# B&R Automation Studio project TD52 (part 20)

### rtmmacros.h
```c
/*
 * Copyright 1994-2005 The MathWorks, Inc.
 *
 * File: rtmmacros.h     $Revision: 1.6.4.9 $
 *
 * Abstract:
 * All our real-time simulation wrappers are setup to handle rtModel
 * objects. For targets that still use the SimStruct, this file
 * provides a mapping from the rtModel to the SimStruct. When all targets
 * use the rtModel, this file can be eliminated.
 */

#ifndef _RTW_HEADER_rtmmacros_h_
# define _RTW_HEADER_rtmmacros_h_

#define rtmGetBlkStateChange            ssGetBlkStateChange
#define rtmSetBlkStateChange            ssSetBlkStateChange
#define rtmGetChecksum0                 ssGetChecksum0
#define rtmSetChecksum0                 ssSetChecksum0
#define rtmGetChecksum1                 ssGetChecksum1
#define rtmSetChecksum1                 ssSetChecksum1
#define rtmGetChecksum2                 ssGetChecksum2
#define rtmSetChecksum2                 ssSetChecksum2
#define rtmGetChecksum3                 ssGetChecksum3
#define rtmSetChecksum3                 ssSetChecksum3
#define rtmGetNumSampleTimes            ssGetNumSampleTimes
#define rtmGetNumContStates             ssGetNumContStates
#define rtmGetContStates                ssGetContStates
#define rtmSetContStates                ssSetContStates
#define rtmIsContinuousTask             ssIsContinuousTask
#define rtmGetDerivCacheNeedsReset      ssGetDerivCacheNeedsReset
#define rtmSetDerivCacheNeedsReset      ssSetDerivCacheNeedsReset
#define rtmGetDiscStates                ssGetDiscStates
#define rtmSetDiscStates                ssSetDiscStates
#define rtmGetErrorStatus               ssGetErrorStatus
#define rtmSetErrorStatus               ssSetErrorStatus
#define rtmGetFixedStepSize             ssGetFixedStepSize
#define rtmSetFixedStepSize             ssSetFixedStepSize
#define rtmGetRTWLogInfo                ssGetRTWLogInfo
#define rtmSetRTWLogInfo                ssSetRTWLogInfo
#define rtmGetRTWExtModeInfo            ssGetRTWExtModeInfo
#define rtmSetRTWExtModeInfo            ssSetRTWExtModeInfo
#define rtmGetMaxNumMinSteps            ssGetMaxNumMinSteps
#define rtmSetMaxNumMinSteps            ssSetMaxNumMinSteps
#define rtmGetMaxStepSize               ssGetMaxStepSize
#define rtmSetMaxStepSize               ssSetMaxStepSize
#define rtmGetMinStepSize               ssGetMinStepSize
#define rtmSetMinStepSize               ssSetMinStepSize
#define rtmGetSolverMaxConsecutiveMinStep   ssGetSolverMaxConsecutiveMinStep
#define rtmSetSolverMaxConsecutiveMinStep   ssSetSolverMaxConsecutiveMinStep
#define rtmGetSolverZcThreshold         ssGetSolverZcThreshold
#define rtmSetSolverZcThreshold         ssSetSolverZcThreshold
#define rtmGetSolverConsecutiveZCsError     ssGetSolverConsecutiveZCsError
#define rtmSetSolverConsecutiveZCsError     ssSetSolverConsecutiveZCsError
#define rtmGetSolverZeroCrossAlgorithm  ssGetSolverZeroCrossAlgorithm
#define rtmSetSolverZeroCrossAlgorithm  ssSetSolverZeroCrossAlgorithm
#define rtmGetSolverShapePreserveControl   ssGetSolverShapePreserveControl
#define rtmSetSolverShapePreserveControl   ssSetSolverShapePreserveControl
#define rtmGetModelMappingInfo          ssGetModelMappingInfo
#define rtmSetModelMappingInfo          ssSetModelMappingInfo
#define rtmGetOffsetTimePtr             ssGetOffsetTimePtr
#define rtmSetOffsetTimePtr             ssSetOffsetTimePtr
#define rtmGetPerTaskSampleHitsPtr      ssGetPerTaskSampleHitsPtr
#define rtmSetPerTaskSampleHitsPtr      ssSetPerTaskSampleHitsPtr
#define rtmIsSampleHit                  ssIsSampleHit
#define rtmSetSampleHitInTask           ssSetSampleHitInTask
#define rtmGetSampleHitPtr              ssGetSampleHitPtr
#define rtmSetSampleHitPtr              ssSetSampleHitPtr
#define rtmGetSampleTime                ssGetSampleTime
#define rtmSetSampleTime                ssSetSampleTime
#define rtmGetSampleTimePtr             ssGetSampleTimePtr
#define rtmSetSampleTimePtr             ssSetSampleTimePtr
#define rtmGetSampleTimeTaskIDPtr       ssGetSampleTimeTaskIDPtr
#define rtmSetSampleTimeTaskIDPtr       ssSetSampleTimeTaskIDPtr
#define rtmGetSimMode                   ssGetSimMode
#define rtmSetSimMode                   ssSetSimMode
#define rtmGetSimTimeStep               ssGetSimTimeStep
#define rtmSetSimTimeStep               ssSetSimTimeStep
#define rtmGetSolverAbsTol              ssGetSolverAbsTol
#define rtmSetSolverAbsTol              ssSetSolverAbsTol
#define rtmGetSolverData                ssGetSolverData
#define rtmSetSolverData                ssSetSolverData
#define rtmGetSolverMaxOrder            ssGetSolverMaxOrder
#define rtmSetSolverMaxOrder            ssSetSolverMaxOrder
#define rtmGetSolverConsecutiveZCsStepRelTol   ssGetSolverConsecutiveZCsStepRelTol
#define rtmSetSolverConsecutiveZCsStepRelTol   ssSetSolverConsecutiveZCsStepRelTol
#define rtmGetSolverMaxConsecutiveZCs   ssGetSolverMaxConsecutiveZCs
#define rtmSetSolverMaxConsecutiveZCs   ssSetSolverMaxConsecutiveZCs
#define rtmGetSolverExtrapolationOrder  ssGetSolverExtrapolationOrder
#define rtmSetSolverExtrapolationOrder  ssSetSolverExtrapolationOrder
#define rtmGetSolverNumberNewtonIterations   ssGetSolverNumberNewtonIterations
#define rtmSetSolverNumberNewtonIterations   ssSetSolverNumberNewtonIterations
#define rtmGetSolverMode                ssGetSolverMode
#define rtmSetSolverMode                ssSetSolverMode
#define rtmGetSolverName                ssGetSolverName
#define rtmSetSolverName                ssSetSolverName
#define rtmGetSolverNeedsReset          ssGetSolverNeedsReset
#define rtmSetSolverNeedsReset          ssSetSolverNeedsReset
#define rtmGetSolverRefineFactor        ssGetSolverRefineFactor
#define rtmSetSolverRefineFactor        ssSetSolverRefineFactor
#define rtmGetSolverRelTol              ssGetSolverRelTol
#define rtmSetSolverRelTol              ssSetSolverRelTol
#define rtmGetSolverStopTime            ssGetSolverStopTime
#define rtmSetSolverStopTime            ssSetSolverStopTime
#define rtmGetSolverRobustResetMethod   ssGetSolverRobustResetMethod
#define rtmSetSolverRobustResetMethod   ssSetSolverRobustResetMethod
#define rtmIsSpecialSampleHit           ssIsSpecialSampleHit
#define rtmGetStepSize                  ssGetStepSize
#define rtmSetStepSize                  ssSetStepSize
#define rtmGetStopRequested             ssGetStopRequested
#define rtmSetStopRequested             ssSetStopRequested
#define rtmGetT                         ssGetT
#define rtmSetT                         ssSetT
#define rtmGetTFinal                    ssGetTFinal
#define rtmSetTFinal                    ssSetTFinal
#define rtmGetTPtr                      ssGetTPtr
#define rtmSetTPtr                      ssSetTPtr
#define rtmGetTStart                    ssGetTStart
#define rtmSetTStart                    ssSetTStart
#define rtmGetTaskTime                  ssGetTaskTime
#define rtmSetTaskTime                  ssSetTaskTime
#define rtmGetTimeOfLastOutput          ssGetTimeOfLastOutput
#define rtmSetTimeOfLastOutput          ssSetTimeOfLastOutput
#define rtmGetTimingData                ssGetTimingData
#define rtmSetTimingData                ssSetTimingData
#define rtmGetU                         ssGetU
#define rtmSetU                         ssSetU
#define rtmGetVariableStepSolver        ssGetVariableStepSolver
#define rtmSetVariableStepSolver        ssSetVariableStepSolver
#define rtmGetY                         ssGetY
#define rtmSetY                         ssSetY
#define rtmGetZCCacheNeedsReset         ssGetZCCacheNeedsReset
#define rtmSetZCCacheNeedsReset         ssSetZCCacheNeedsReset
#define rtmGetdX                        ssGetdX
#define rtmSetdX                        ssSetdX
#define rtmOutputs                      sfcnOutputs
#define rtmTerminate                    sfcnTerminate
#define rtmInitializeSampleTimes        sfcnInitializeSampleTimes
#define rtmInitializeSizes              sfcnInitializeSizes
#define rtmUpdate                       sfcnUpdate
#define rtmDerivatives                  sfcnDerivatives
#define rtmStart                        sfcnStart
#endif                                  /* _RTW_HEADER_rtmmacros_h_ */

/* [EOF] rtmmacros.h */
```

### rtsplntypes.h
```c
#ifndef RTSPLNTYPES_H
#define RTSPLNTYPES_H

/*
 * File: rtsplntypes.h
 *
 * Abstract:
 *
 *   Typedefs for spline lookup table algorithms.
 *
 *   Copyright 1994-2007 The MathWorks, Inc.
 *
 *   $Revision: 1.1.6.1 $
 *
 */

#include "rtwtypes.h"

/***************************************************************
 *                n-D Table Work Data Structures               *
 ***************************************************************/

typedef struct rt_LUTnWork_tag
{
    const uint32_T *m_dimSizes;
    void           *m_tableData;
    void           **m_bpDataSet;
    uint32_T       *m_bpIndex;
    void           *m_bpLambda;
    const uint32_T *m_maxIndex;
} rt_LUTnWork;

typedef struct rt_LUTSplineWork_tag
{
    rt_LUTnWork    *m_TWork;
    void           *m_yyA;
    void           *m_yyB;
    void           *m_yy2;
    void           *m_up;
    void           *m_y2;
    const uint32_T *m_numYWorkElts;
} rt_LUTSplineWork;

#endif  /* RTSPLNTYPES_H */
```

### rtw_capi.h
```c
/*
 * Copyright 1994-2008 The MathWorks, Inc.
 *
 * File: rtw_capi.h     $Revision $
 *
 * Abstract:
 *   Provides structure types and constants generated by CAPI.
 *   Macros for accessing the fields of the structures are also provided.
 *   This header file is included in MODEL_capi.c
 *
 */

#ifndef _RTW_CAPI_H_
# define _RTW_CAPI_H_

#include <rtwtypes.h>

#define SS_ENUM_TYPE (MAX_uint8_T-1)
#define SS_STRUCT    (MAX_uint8_T)
#define rt_offsetof(s,el) ((uint16_T)((char_T *)&((s *)0)->el - (char_T *)(s *)0))

/* Enumeration for fixed point scaling type*/
typedef enum {
  rtwCAPI_FIX_UNIFORM_SCALING,
  rtwCAPI_FIX_NONUNIFORM_SCALING,
  rtwCAPI_FIX_RESERVED
} rtwCAPI_FixPtScalingType;

/* Enumeration for data orientation */
typedef enum {
  rtwCAPI_SCALAR,
  rtwCAPI_VECTOR,
  rtwCAPI_MATRIX_ROW_MAJOR,
  rtwCAPI_MATRIX_COL_MAJOR,
  rtwCAPI_MATRIX_COL_MAJOR_ND
} rtwCAPI_Orientation;

/* Signals Structure */
/* Fields of this stucture can be used to monitor block output signals*/
typedef struct rtwCAPI_Signals_tag {
  uint_T    addrMapIndex;  /* index into the data address map                */
  uint_T    sysNum;        /* system identification number, where 0 = root   */
  const char_T *blockPath; /* block's full path name (RTW mangled version)   */
  const char_T *signalName;/* signal label (unmangled, NULL if not present)  */
  uint16_T  portNumber;    /* port number  (starts at 0)                     */
  uint16_T  dataTypeIndex; /* index into DataTypeMap, gives signal data type */
  uint16_T  dimIndex;      /* index into DimensionMap, gives signal dimension*/
  uint16_T  fxpIndex;      /* index into FixPtMap, gives Fixed point info    */
  uint8_T   sTimeIndex;    /* index into SampleTimeMap, gives Task info      */
} rtwCAPI_Signals;

/* Macros for accessing Signals structure fields */
/* bio is a pointer to array of Signals structures */
#define rtwCAPI_GetSignalAddrIdx(bio, i)       ((bio)[(i)].addrMapIndex)
#define rtwCAPI_GetSignalBlockPath(bio, i)     ((bio)[(i)].blockPath)
#define rtwCAPI_GetSignalName(bio, i)          ((bio)[(i)].signalName)
#define rtwCAPI_GetSignalPortNumber(bio, i)    ((bio)[(i)].portNumber)
#define rtwCAPI_GetSignalDataTypeIdx(bio, i)   ((bio)[(i)].dataTypeIndex)
#define rtwCAPI_GetSignalDimensionIdx(bio, i)  ((bio)[(i)].dimIndex)
#define rtwCAPI_GetSignalFixPtIdx(bio, i)      ((bio)[(i)].fxpIndex)
#define rtwCAPI_GetSignalSampleTimeIdx(bio, i) ((bio)[(i)].sTimeIndex)
#define rtwCAPI_GetSignalSysNum(bio, i)        ((bio)[(i)].sysNum)

/* BlockParameters Structure */
/* Fields of this structure can be used to monitor/modify block parameters */
typedef struct rtwCAPI_BlockParameters_tag {
  uint_T    addrMapIndex;  /* index into the data address map                */
  const char_T *blockPath; /* block's full path name (RTW mangled version)   */
  const char_T *paramName; /* parameter name                                 */
  uint16_T  dataTypeIndex; /* index into DataTypeMap, gives param data type  */
  uint16_T  dimIndex;      /* index into DimensionMap, gives param dimensions*/
  uint16_T  fxpIndex;      /* index into FixPtMap, gives Fixed point info    */
} rtwCAPI_BlockParameters;

/* Macros for accessing BlockParameter structure fields */
/* prm is a pointer to array of BlockParameter structures */
#define rtwCAPI_GetBlockParameterAddrIdx(prm, i)      ((prm)[(i)].addrMapIndex)
#define rtwCAPI_GetBlockParameterBlockPath(prm, i)    ((prm)[(i)].blockPath)
#define rtwCAPI_GetBlockParameterName(prm, i)         ((prm)[(i)].paramName)
#define rtwCAPI_GetBlockParameterDataTypeIdx(prm, i)  ((prm)[(i)].dataTypeIndex)
#define rtwCAPI_GetBlockParameterDimensionIdx(prm, i) ((prm)[(i)].dimIndex)
#define rtwCAPI_GetBlockParameterFixPtIdx(prm, i)     ((prm)[(i)].fxpIndex)

/* ModelParameter Structure */
/* Fields of this structure can be used to monitor/modify model parameters   *
 * When Inline Parameters is on, you can configure tunable block parameters  *
 * as model parameters.                                                      */
typedef struct rtwCAPI_ModelParameters_tag {
  uint_T    addrMapIndex;  /* index into the data address map                */
  const char_T   *varName; /* variable  name                                 */
  uint16_T  dataTypeIndex; /* index into DataTypeMap, gives param data type  */
  uint16_T  dimIndex;      /* index into DimensionMap, gives param dimensions*/
  uint16_T  fxpIndex;      /* index into FixPtMap, gives Fixed point info    */
} rtwCAPI_ModelParameters;

/* Macros for accessing ModelParameter structure fields */
/* prm is a pointer to array of ModelParameter structures */
#define rtwCAPI_GetModelParameterAddrIdx(prm, i)      ((prm)[(i)].addrMapIndex)
#define rtwCAPI_GetModelParameterName(prm, i)         ((prm)[(i)].varName)
#define rtwCAPI_GetModelParameterDataTypeIdx(prm, i)  ((prm)[(i)].dataTypeIndex)
#define rtwCAPI_GetModelParameterDimensionIdx(prm, i) ((prm)[(i)].dimIndex)
#define rtwCAPI_GetModelParameterFixPtIdx(prm, i)     ((prm)[(i)].fxpIndex)

/* rtwCAPI_States Structure */
/* Fields of this stucture can be used to monitor block States */
typedef struct rtwCAPI_States_tag {
  uint_T addrMapIndex;     /* index into the data address map                 */
  int_T  contStateStartIndex; /* starting index in the model's continuous     *
                               * state and state derivative vectors. This is  *
                               * set to -1 for discrete states                */
  const char_T *blockPath; /* block's full path name (RTW mangled version)    */
  const char_T *stateName; /* state name, Default:DWork/Cont State Identifier */
  const char_T *pathAlias; /* Alias block path */
  uint16_T  dWorkIndex;    /* Index into the Block DWork, 0 for cont. states  */
  uint16_T  dataTypeIndex; /* index into DataTypeMap, gives state data type   */
  uint16_T  dimIndex;      /* index into DimensionMap, gives state dimensions */
  uint16_T  fxpIndex;      /* index into FixPtMap, gives Fixed point info     */
  uint8_T   sTimeIndex;    /* index into SampleTimeMap, gives Task info       */
  uint8_T   isContinuous;  /* if the state is a Continuous state*/
} rtwCAPI_States;

/* Macros for accessing States structure fields */
/* bState is a pointer to array of States structures */
#define rtwCAPI_GetStateAddrIdx(bState, i)       ((bState)[(i)].addrMapIndex)
#define rtwCAPI_GetContStateStartIndex(bState, i) \
        ((bState)[(i)].contStateStartIndex)
#define rtwCAPI_GetStateBlockPath(bState, i)     ((bState)[(i)].blockPath)
#define rtwCAPI_GetStateName(bState, i)          ((bState)[(i)].stateName)
#define rtwCAPI_GetStatePathAlias(bState, i)     ((bState)[(i)].pathAlias)
#define rtwCAPI_GetStateDWorkIdx(bState, i)      ((bState)[(i)].dWorkIndex)
#define rtwCAPI_GetStateDataTypeIdx(bState, i)   ((bState)[(i)].dataTypeIndex)
#define rtwCAPI_GetStateDimensionIdx(bState, i)  ((bState)[(i)].dimIndex)
#define rtwCAPI_GetStateFixPtIndex(bState, i)    ((bState)[(i)].fxpIndex)
#define rtwCAPI_GetStateSampleTimeIdx(bState, i) ((bState)[(i)].sTimeIndex)
#define rtwCAPI_IsAContinuousState(bState, i)    ((bState)[(i)].isContinuous == 1)

/* DataTypeMap structure */
/* Members provide data type information of a signal or parameter */
typedef struct rtwCAPI_DataTypeMap_tag {
  const char_T *cDataName;   /* C language data type name                    */
  const char_T *mwDataName;  /* MathWorks data type, typedef in rtwtypes.h   */
  uint16_T      numElements; /* number of elements, 0 for non-structure data */
  uint16_T      elemMapIndex;/* index into the ElementMap, gives Bus Info    */
  uint16_T      dataSize;    /* data size in Bytes                           */
  uint8_T       slDataId;    /* enumerated data type from simstruc_types.h   */
  unsigned int  isComplex:1; /* is the data type complex (1=Complex, 0=Real) */
  unsigned int  isPointer:1; /* is data accessed Via Pointer (1=yes, 0= no)  */
} rtwCAPI_DataTypeMap;

/* Notes on rtwCAPI_DataTypeMap:
 * cDataName  - The ANSI C equivalent data type.
 *              For fixed point data
 *                  cDataName = the native integer equivalent
 *              For Complex data or non-virtual structures,
 *                  cDataName = "struct"
 * mwDataName - RTW defined data type. Typedef can be found in rtwtypes.h
 *              For fixed point data,
 *                  mwDataName = the integer type in which the data is stored.
 *                  Use rtwCAPI_FixPtMap to get slope & bias of the data.
 * numElements - Number of elements/members in the data type. If the data type
 *              represents a non-virtual structure (for e.g, bus structure),
 *              this field gives the number of elements in the structure.
 *              For non-structure data type, the default value is 0
 *              Complex data types are treated as non-structures
 * elemMapIndex - Index into the rtwCAPI_ElementMap which maps each of the
 *              element/member of a structure data type.
 * slDataId   - Enumerated Simulink Data type defined in simstruc_types.h.
 *              The enumerations are
 *                 o SS_DOUBLE
 *                 o SS_SINGLE
 *                 o SS_INT8
 *                 o SS_UINT8
 *                 o SS_INT16
 *                 o SS_UINT16
 *                 o SS_INT32
 *                 o SS_UINT32
 *                 o SS_BOOLEAN
 *                 o SS_ENUM_TYPE  (for enumerated data types)
 *                 o SS_STRUCT     (for non-virtual structures)
 *              For fixed point data:
 *                  slDataId = enumeration corresponding to the integer type
 *                             in which the data is stored
 *              For Complex data:
 *                  slDataId = enumeration corresponding to the data type of
 *                             the real part.
 * isComplex  - is the data type complex (1=Complex, 0=Real)
 * isPointer  - is data accessed Via Pointer (1=yes, 0= no)
 */

/* Macros for accessing DataTypeMap fields/members */
#define rtwCAPI_GetDataTypeCName(dTypeMap, i)       ((dTypeMap)[(i)].cDataName)
#define rtwCAPI_GetDataTypeMWName(dTypeMap, i)      ((dTypeMap)[(i)].mwDataName)
#define rtwCAPI_GetDataTypeNumElements(dTypeMap, i) ((dTypeMap)[(i)].numElements)
#define rtwCAPI_GetDataTypeElemMapIndex(dTypeMap,i) ((dTypeMap)[(i)].elemMapIndex)
#define rtwCAPI_GetDataTypeSLId(dTypeMap, i)        ((dTypeMap)[(i)].slDataId)
#define rtwCAPI_GetDataTypeSize(dTypeMap, i)        ((dTypeMap)[(i)].dataSize)
#define rtwCAPI_GetDataIsComplex(dTypeMap, i)       ((dTypeMap)[(i)].isComplex)
#define rtwCAPI_GetDataIsPointer(dTypeMap, i)       ((dTypeMap)[(i)].isPointer)

/* Macros for determining whether signals/states support MAT-File logging */
#define rtwCAPI_CanLogSignalToMATFile(dTypeMap, bio, i) \
    (rtwCAPI_GetDataTypeSLId(dTypeMap, rtwCAPI_GetSignalDataTypeIdx(bio, i))   < SS_NUM_BUILT_IN_DTYPE)
#define rtwCAPI_CanLogStateToMATFile(dTypeMap, bState, i) \
    (rtwCAPI_GetDataTypeSLId(dTypeMap, rtwCAPI_GetStateDataTypeIdx(bState, i)) < SS_NUM_BUILT_IN_DTYPE)

/* ElementMap structure */
/* Fields provide information on elements (fields) in Simulink Bus structure */
typedef struct rtwCAPI_ElementMap_tag {
  const char_T   *elementName;   /* name of the element                      */
  uint16_T  elementOffset; /* offset of the structure element in bytes       */
  uint16_T  dataTypeIndex; /* index into DataTypeMap, datatype of the element*/
  uint16_T  dimIndex;      /* index into DimensionMap, element's dimensions  */
  uint16_T  fxpIndex;      /* index into fixPtMap, fixed point information   */
} rtwCAPI_ElementMap;

/* Macros for accessing ElementMap fields */
#define rtwCAPI_GetElementName(elemMap, i)         ((elemMap)[(i)].elementName)
#define rtwCAPI_GetElementOffset(elemMap, i)       ((elemMap)[(i)].elementOffset)
#define rtwCAPI_GetElementDataTypeIdx(elemMap, i)  ((elemMap)[(i)].dataTypeIndex)
#define rtwCAPI_GetElementDimensionIdx(elemMap, i) ((elemMap)[(i)].dimIndex)
#define rtwCAPI_GetElementFixPtIdx(elemMap, i)     ((elemMap)[(i)].fxpIndex)

/* DimensionMap structure */
/* Fields provide dimensions of a signal or a parameter */
typedef struct rtwCAPI_DimensionMap_tag {
  rtwCAPI_Orientation orientation;
                                 /* orientation of data -scalar/vector/matrix/ND */
  uint_T    dimArrayIndex;       /* index into dimension array                   */
  uint8_T   numDims;             /* number of dimensions                         */
  uint_T    vardimsIndex;        /* index into vardims address array             */
} rtwCAPI_DimensionMap;

/* Macros for accessing DimensionMap fields */
#define rtwCAPI_GetOrientation(dimMap, i)    ((dimMap)[(i)].orientation)
#define rtwCAPI_GetDimArrayIndex(dimMap, i)  ((dimMap)[(i)].dimArrayIndex)
#define rtwCAPI_GetNumDims(dimMap, i)        ((dimMap)[(i)].numDims)
#define rtwCAPI_GetDimsIsVariable(vardimsAddrMap, dimMap, i) (vardimsAddrMap[(dimMap)[(i)].vardimsIndex] != NULL)

/* FixPtMap Structure */
/* Fields provide fixed point information of a signal or parameter */
typedef struct rtwCAPI_FixPtMap_tag {
  const void*       fracSlopePtr;   /* pointer to fractional slope value        */
  const void*       biasPtr;        /* pointer to bias value                    */
  rtwCAPI_FixPtScalingType scaleType;
                              /* scaling type - uniform/non-uniform       */
  uint8_T     wordLength;     /* number of bits required to store value   *
                               * In MATLAB, word length of the fi object  */
  int8_T      exponent;       /* exponent                                 */
  boolean_T   isSigned;       /* 1 = signed data, 0 = unsigned data       */
} rtwCAPI_FixPtMap;

/* Macros for accessing FixPtMap fields */
#define rtwCAPI_GetFxpFracSlopePtr(fxpMap, i) ((fxpMap)[(i)].fracSlopePtr)
#define rtwCAPI_GetFxpBiasPtr(fxpMap, i)      ((fxpMap)[(i)].biasPtr)
#define rtwCAPI_GetFxpScaling(fxpMap, i)      ((fxpMap)[(i)].scaleType)
#define rtwCAPI_GetFxpWordLength(fxpMap, i)   ((fxpMap)[(i)].wordLength)
#define rtwCAPI_GetFxpExponent(fxpMap, i)     ((fxpMap)[(i)].exponent)
#define rtwCAPI_GetFxpIsSigned(fxpMap, i)     ((fxpMap)[(i)].isSigned)

/* Macros to get the slope and bias values casted to DOUBLE */
#define rtwCAPI_GetFxpFracSlope(fxpMap, i) (*((real_T*) rtwCAPI_GetFxpFracSlopePtr(fxpMap,i)))
#define rtwCAPI_GetFxpBias(fxpMap, i)      (*((real_T*) rtwCAPI_GetFxpBiasPtr(fxpMap, i)))

/* SampleTimeMap Structure */
typedef struct rtwCAPI_SampleTimeMap_tag {
  const void*     samplePeriodPtr;  /* pointer to sample time period value       */
  const void*     sampleOffsetPtr;  /* pointer to sample time Offset value       */
  int8_T    tid;              /* task identifier                           */
  uint8_T   samplingMode;     /* 1 = FrameBased, 0 = SampleBased           */
} rtwCAPI_SampleTimeMap;

/* Macros for accessing SampleTimeMap fields */

#define rtwCAPI_GetSamplePeriodPtr(sampTimeMap, i) ((sampTimeMap)[(i)].samplePeriodPtr)
#define rtwCAPI_GetSampleOffsetPtr(sampTimeMap, i) ((sampTimeMap)[(i)].sampleOffsetPtr)
#define rtwCAPI_GetSampleTimeTID(sampTimeMap, i)   ((sampTimeMap)[(i)].tid)
#define rtwCAPI_GetSamplingMode(sampTimeMap, i)    ((sampTimeMap)[(i)].samplingMode)

/* Macros to get sample period and offset casted to DOUBLE */
#define rtwCAPI_GetSamplePeriod(sampTimeMap, i) (*((real_T *) rtwCAPI_GetSamplePeriodPtr(sampTimeMap, i)))
#define rtwCAPI_GetSampleOffset(sampTimeMap, i) (*((real_T *) rtwCAPI_GetSampleOffsetPtr(sampTimeMap, i)))

/* Macro to get the actual data address */
#define rtwCAPI_GetDataAddress(dataAddrMap,addrIdx) ((dataAddrMap)[(addrIdx)])

/* Macro to get the actual var dims address */
#define rtwCAPI_GetCurrentDimsAddr(vardimsAddrMap,dimMap,addrIdx) ((vardimsAddrMap)[(dimMap)[(addrIdx)].vardimsIndex])

#endif /* _RTW_CAPI_H_ */

/* EOF - rtw_capi.h */
```

### rtw_capi_examples.h
```c
/*
 * Copyright 2004 The MathWorks, Inc.
 *
 * File: rtw_capi_examples.h     $Revision: 1.1.4.2 $
 *
 * Abstract:
 *   Provides utility functions to traverse and access RTW generated C-API
 *   structures. The C-API structure types are provided in following 2 files.
 *
 *       matlabroot/rtw/c/src/rtw_capi.h & rtw_modelmap.h
 *
 *   The actual data structures are generated by code generator in
 *   <MODEL>_capi.c, where <MODEL> is the name of the model.
 *
 *   The functions provided in this file are
 *       capi_PrintModelParameter - Prints a model parameter value to STDOUT
 */

#ifndef __RTW_CAPI_EXAMPLES_H__
# define __RTW_CAPI_EXAMPLES_H__

#include <stdio.h>
#include <assert.h>
#include <math.h>
#include "rtwtypes.h"
#include "rtw_modelmap.h"

#ifdef __cplusplus
extern "C" {
#endif

extern void capi_PrintModelParameter(rtwCAPI_ModelMappingInfo* capiMap,
                                     uint_T                    paramIdx);

extern void capi_PrintParameter(const char_T*  paramName,
                                void*          paramAddress,
                                uint8_T        slDataId,
                                unsigned short isComplex,
                                uint_T*        actDims,
                                uint_T         numDims,
                                real_T         slope,
                                real_T         bias);

extern int_T capi_ModifyModelParameter(rtwCAPI_ModelMappingInfo* capiMap,
                                       uint_T                    paramIdx,
                                       void*                     newParam);

extern int_T capi_ModifyParameter(void                 *_param,
                                  void                 *_newParam,
                                  rtwCAPI_Orientation  orientation,
                                  uint_T               *dims,
                                  uint8_T              nDims,
                                  uint8_T              slDataType,
                                  unsigned short       isComplex);

#ifdef __cplusplus
}
#endif

#endif

/* EOF - rtw_capi_example.h */
```

### rtw_continuous.h
```c
/*
 * Copyright 1990-2009 The MathWorks, Inc.
 *
 * File: rtw_continuous.h     $Revision: 1.1.6.3 $
 *
 * Abstract:
 *   Type definitions for continuous-time support.
 *
 */

#ifndef __RTW_CONTINUOUS_H__
#define __RTW_CONTINUOUS_H__

/* For models registering MassMatrix */
typedef enum {
    SS_MATRIX_NONE,
    SS_MATRIX_CONSTANT,
    SS_MATRIX_TIMEDEP,
    SS_MATRIX_STATEDEP
} ssMatrixType;

typedef enum {
    SOLVER_MODE_AUTO,          /* only occurs in
                                  mdlInitializeSizes/mdlInitializeSampleTimes */
    SOLVER_MODE_SINGLETASKING,
    SOLVER_MODE_MULTITASKING
} SolverMode;

typedef enum {
    MINOR_TIME_STEP,
    MAJOR_TIME_STEP
} SimTimeStep;

/* =============================================================================
 * Model methods object
 * =============================================================================
 */
typedef void (*rtMdlInitializeSizesFcn)(void *rtModel);
typedef void (*rtMdlInitializeSampleTimesFcn)(void *rtModel);
typedef void (*rtMdlStartFcn)(void *rtModel);
typedef void (*rtMdlOutputsFcn)(void *rtModel, int_T tid);
typedef void (*rtMdlUpdateFcn)(void *rtModel, int_T tid);
typedef void (*rtMdlDerivativesFcn)(void *rtModel);
typedef void (*rtMdlProjectionFcn)(void *rtModel);
typedef void (*rtMdlMassMatrixFcn)(void *rtModel);
typedef void (*rtMdlForcingFunctionFcn)(void *rtModel);
typedef void (*rtMdlTerminateFcn)(void *rtModel);
#ifdef RT_MALLOC
typedef real_T (*rtMdlDiscreteEventsFcn)(void  *pModel,
                                         int_T  rtmNumSampTimes,
                                         void  *rtmTimingData,
                                         int_T  *rtmSampleHitPtr,
                                         int_T  *rtmPerTaskSampleHits);
#endif

typedef struct _RTWRTModelMethodsInfo_tag {
    void                          *rtModelPtr;
    rtMdlInitializeSizesFcn       rtmInitSizesFcn;
    rtMdlInitializeSampleTimesFcn rtmInitSampTimesFcn;
    rtMdlStartFcn                 rtmStartFcn;
    rtMdlOutputsFcn               rtmOutputsFcn;
    rtMdlUpdateFcn                rtmUpdateFcn;
    rtMdlDerivativesFcn           rtmDervisFcn;
    rtMdlProjectionFcn            rtmProjectionFcn;
    rtMdlMassMatrixFcn            rtmMassMatrixFcn;
    rtMdlForcingFunctionFcn       rtmForcingFunctionFcn;
    rtMdlTerminateFcn             rtmTerminateFcn;
#ifdef  RT_MALLOC
    rtMdlDiscreteEventsFcn        rtmDiscreteEventsFcn;
#endif
} RTWRTModelMethodsInfo;

#define rtmiSetRTModelPtr(M,rtmp) ((M).rtModelPtr = (rtmp))
#define rtmiGetRTModelPtr(M)      (M).rtModelPtr

#define rtmiSetInitSizesFcn(M,fp) \
  ((M).rtmInitSizesFcn = ((rtMdlInitializeSizesFcn)(fp)))
#define rtmiSetInitSampTimesFcn(M,fp) \
  ((M).rtmInitSampTimesFcn = ((rtMdlInitializeSampleTimesFcn)(fp)))
#define rtmiSetStartFcn(M,fp) \
  ((M).rtmStartFcn = ((rtMdlStartFcn)(fp)))
#define rtmiSetOutputsFcn(M,fp) \
  ((M).rtmOutputsFcn = ((rtMdlOutputsFcn)(fp)))
#define rtmiSetUpdateFcn(M,fp) \
  ((M).rtmUpdateFcn = ((rtMdlUpdateFcn)(fp)))
#define rtmiSetDervisFcn(M,fp) \
  ((M).rtmDervisFcn = ((rtMdlDerivativesFcn)(fp)))
#define rtmiSetProjectionFcn(M,fp) \
  ((M).rtmProjectionFcn = ((rtMdlProjectionFcn)(fp)))
#define rtmiSetMassMatrixFcn(M,fp) \
  ((M).rtmMassMatrixFcn = ((rtMdlMassMatrixFcn)(fp)))
#define rtmiSetForcingFunctionFcn(M,fp) \
  ((M).rtmForcingFunctionFcn = ((rtMdlForcingFunctionFcn)(fp)))
#define rtmiSetTerminateFcn(M,fp) \
  ((M).rtmTerminateFcn = ((rtMdlTerminateFcn)(fp)))
#ifdef  RT_MALLOC
#define rtmiSetDiscreteEventsFcn(M,fp) \
  ((M).rtmDiscreteEventsFcn = ((rtMdlDiscreteEventsFcn)(fp)))
#endif

#define rtmiInitializeSizes(M)                  \
    ((*(M).rtmInitSizesFcn)((M).rtModelPtr))
#define rtmiInitializeSampleTimes(M)                    \
    ((*(M).rtmInitSampTimesFcn)((M).rtModelPtr))
#define rtmiStart(M) \
    ((*(M).rtmStartFcn)((M).rtModelPtr))
#define rtmiOutputs(M, tid) \
    ((*(M).rtmOutputsFcn)((M).rtModelPtr,tid))
#define rtmiUpdate(M, tid) \
    ((*(M).rtmUpdateFcn)((M).rtModelPtr,tid))
#define rtmiDerivatives(M) \
    ((*(M).rtmDervisFcn)((M).rtModelPtr))
#define rtmiProjection(M) \
    ((*(M).rtmProjectionFcn)((M).rtModelPtr))
#define rtmiMassMatrix(M) \
    ((*(M).rtmMassMatrixFcn)((M).rtModelPtr))
#define rtmiForcingFunction(M) \
    ((*(M).rtmForcingFunctionFcn)((M).rtModelPtr))
#define rtmiTerminate(M) \
    ((*(M).rtmTerminateFcn)((M).rtModelPtr))
#ifdef  RT_MALLOC
#define rtmiDiscreteEvents(M,x1,x2,x3,x4)                               \
    ((*(M).rtmDiscreteEventsFcn)((M).rtModelPtr,(x1),(x2),(x3),(x4)))
#endif
#endif /* __RTW_CONTINUOUS_H__ */
```

### rtw_extmode.h
```c
/*
 * Copyright 1990-2008 The MathWorks, Inc.
 *
 * File: rtw_extmode.h     $Revision: 1.1.6.3 $
 *
 * Abstract:
 *   Type definitions for Simulink External Mode support.
 */

#ifndef __RTW_EXTMODE_H__
#define __RTW_EXTMODE_H__

/* =============================================================================
 * External mode object
 * =============================================================================
 */
typedef struct _RTWExtModeInfo_tag {

    void *subSysActiveVectorAddr;  /* Array of addresses pointing to
                                    * the active vector slots for sub-systems.
                                    * Sub-systems store information about their
                                    * state in their extmode active vector.
                                    */
    uint32_T *checksumsPtr;        /* Pointer to the model's checksums array
                                    */
    const void **mdlMappingInfoPtr;/* Pointer to the model's mapping info
                                    * pointer
                                    */

#if !defined(ENABLE_SLEXEC_SSBRIDGE)
    void       *tPtr;              /* Copy of model's time pointer */
#else
    void* simStruct;
#endif

    int32_T tFinalTicks;           /* Used with integer only code, holds the
                                    * number of base rate ticks representing
                                    * the final time (final time in seconds
                                    * divided by base rate step size).
                                    */

} RTWExtModeInfo;

/* gnat 3.12a2 doesn't like use "/" as line continuation here */
#define rteiSetSubSystemActiveVectorAddresses(E,addr) ((E)->subSysActiveVectorAddr = ((void *)addr))
#define rteiGetSubSystemActiveVectorAddresses(E)    ((E)->subSysActiveVectorAddr)
#define rteiGetAddrOfSubSystemActiveVector(E,idx)   ((int8_T*)((int8_T**)((E)->subSysActiveVectorAddr))[idx])

#define rteiSetModelMappingInfoPtr(E,mip) ((E)->mdlMappingInfoPtr = (mip))
#define rteiGetModelMappingInfo(E) (*((E)->mdlMappingInfoPtr))

#define rteiSetChecksumsPtr(E,cp) ((E)->checksumsPtr = (cp))
#define rteiGetChecksum0(E) (E)->checksumsPtr[0]
#define rteiGetChecksum1(E) (E)->checksumsPtr[1]
#define rteiGetChecksum2(E) (E)->checksumsPtr[2]
#define rteiGetChecksum3(E) (E)->checksumsPtr[3]

#if !defined(ENABLE_SLEXEC_SSBRIDGE)
# define rteiSetTPtr(E,p) ((E)->tPtr = (p))
# define rteiGetT(E)      ((time_T *)(E)->tPtr)[0]
#endif

#define rteiGetTFinalTicks(E) ((int32_T)((E)->tFinalTicks))
#define rteiGetPtrTFinalTicks(E) ((int32_T *)(&((E)->tFinalTicks)))

/*
 * UNUSED_PARAMETER(x)
 *   Used to specify that a function parameter (argument) is required but not
 *   accessed by the function body.
 */
#ifndef UNUSED_PARAMETER
# if defined(__LCC__)
#   define UNUSED_PARAMETER(x)  /* do nothing */
# else
/*
 * This is the semi-ANSI standard way of indicating that a
 * unused function parameter is required.
 */
#   define UNUSED_PARAMETER(x) (void) (x)
# endif
#endif

#endif /* __RTW_EXTMODE_H__ */
```

### rtw_linux.h
```c
#ifndef RTW_LINUX_H
#define RTW_LINUX_H

/*
 * Copyright 2011 The MathWorks, Inc.
 *
 * File: rtw_linux.h
 *
 * Abstract:
 *  Function prototypes and defines pthread mutex/semaphores
 */
#include <pthread.h>
#include <stdlib.h>
#include <semaphore.h>

#ifndef __USE_UNIX98
#define __USE_UNIX98
#endif

#ifdef __cplusplus
extern "C" {
#endif

extern void rtw_pthread_mutex_init( void** mutexDW );

#ifdef __cplusplus
}
#endif

#define rtw_pthread_mutex_lock( mutexDW ) \
    pthread_mutex_lock((pthread_mutex_t *)(mutexDW));

#define rtw_pthread_mutex_unlock( mutexDW ) \
    pthread_mutex_unlock((pthread_mutex_t *)(mutexDW));

#define rtw_pthread_mutex_destroy( mutexDW )      \
    pthread_mutex_destroy((pthread_mutex_t *)(mutexDW)); \
    free(mutexDW);

#define rtw_pthread_sem_create( semaphoreDW, initVal ) \
    *semaphoreDW = malloc(sizeof(sem_t));               \
    sem_init(*(semaphoreDW), 0, (initVal));

#define rtw_pthread_sem_wait( semaphoreDW ) \
    sem_wait(semaphoreDW);

#define rtw_pthread_sem_post( semaphoreDW ) \
    sem_post(semaphoreDW);

#define rtw_pthread_sem_destroy( semaphoreDW ) \
    sem_destroy(semaphoreDW);                   \
    free(semaphoreDW);

#endif /* RTW_LINUX_H */

/* LocalWords:  pthread
 */
```

### rtw_linux_mac.h
```c
#ifndef RTW_LINUX_MAC_H
#define RTW_LINUX_MAC_H

/*
 * Copyright 2011 The MathWorks, Inc.
 *
 * File: rtw_linux_mac.h
 *
 * Abstract:
 *  Function prototypes and defines pthread mutex/semaphores
 */
#ifdef __cplusplus
extern "C" {
#endif

#include <pthread.h>
#include <stdlib.h>
#include <semaphore.h>

#ifndef __USE_UNIX98
#define __USE_UNIX98
#endif

extern void rtw_pthread_mutex_init_mac( void** mutexDW );

#define rtw_pthread_mutex_lock_mac( mutexDW )                   \
    pthread_mutex_lock((pthread_mutex_t *)(mutexDW));

#define rtw_pthread_mutex_unlock_mac( mutexDW )                 \
    pthread_mutex_unlock((pthread_mutex_t *)(mutexDW));

#define rtw_pthread_mutex_destroy_mac( mutexDW )                \
    pthread_mutex_destroy((pthread_mutex_t *)(mutexDW));        \
    free(mutexDW);

extern void rtw_pthread_sem_create_mac( void** semaphoreDW1,
                                 void** semaphoreDW2,
                                 long initVal );

#define rtw_pthread_sem_wait_mac( semaphoreDW ) \
    sem_wait(semaphoreDW);

#define rtw_pthread_sem_post_mac( semaphoreDW ) \
    sem_post(semaphoreDW);

#define rtw_pthread_sem_destroy_mac( semaphoreDW ) \
    sem_unlink((char*)(semaphoreDW));              \
    free(semaphoreDW);

#ifdef __cplusplus
}
#endif

#endif /* RTW_LINUX_MAC_H */

/* LocalWords:  pthread
 */
```

### rtw_matlogging.h
```c
/*
 * Copyright 1990-2007 The MathWorks, Inc.
 *
 * File: rtw_matlogging.h     $Revision: 1.1.6.3 $
 *
 * Abstract:
 *   Type definitions for MAT-file logging support.
 */

#ifndef __RTW_MATLOGGING_H__
#define __RTW_MATLOGGING_H__

/*
 * The RTWLogSignalInfo and RTWLogInfo structures are for use by
 * the Real-Time Workshop and should not be used by S-functions.
 */
typedef const int8_T * const * LogSignalPtrsType;

#ifndef NO_FLOATS /* ERT integer-only */

typedef struct RTWLogDataTypeConvert_tag {

    int conversionNeeded;
    BuiltInDTypeId dataTypeIdLoggingTo;
    DTypeId        dataTypeIdOriginal;
    int            bitsPerChunk;
    int            numOfChunk;
    unsigned int   isSigned;
    real_T         fracSlope;
    int            fixedExp;
    real_T         bias;

} RTWLogDataTypeConvert;

typedef struct RTWLogSignalInfo_tag {
    int_T           numSignals;
    int_T          *numCols;
    int_T          *numDims;
    int_T          *dims;
    boolean_T      *isVarDims;       /* Dimension Mode: true -- VarDims / false -- fixed dims */
    void           **currSigDims;    /* current signal dimensions */
    int_T          *currSigDimsSize; /* Size of currSigDims in bytes */
    BuiltInDTypeId *dataTypes;
    int_T          *complexSignals;
    int_T          *frameData;

    union {
        const char_T** cptr;
        char_T**       ptr;
    } labels;

    char_T         *titles;
    int_T          *titleLengths;
    int_T          *plotStyles;

    union {
        const char_T** cptr;
        char_T**       ptr;
    } blockNames;

    union {
        const char_T** cptr;
        char_T**       ptr;
    } stateNames;

    boolean_T      *crossMdlRef;

    RTWLogDataTypeConvert *dataTypeConvert;

} RTWLogSignalInfo;

/* =============================================================================
 * Logging object
 * =============================================================================
 */
typedef struct _RTWLogInfo_tag {
  void              *logInfo;      /* Pointer to a book keeping structure    *
                                    * used in rtwlog.c                       */

  union {
      LogSignalPtrsType cptr; /* Pointers to the memory location    */
      int8_T**    ptr;        /* of the data to be logged into the  *
                               * states structure. Not used if      *
                               * logging data in matrix format.     */

  } logXSignalPtrs;

  union {
      LogSignalPtrsType cptr; /* Pointers to the memory location    */
      int8_T**    ptr;        /* of the data to be logged into the  *
                               * outputs structure. Not used if     *
                               * logging data in matrix format.     */
  } logYSignalPtrs;

  union {
      LogSignalPtrsType cptr; /* Pointers to the memory location    */
      int8_T**    ptr;        /* of the data to be logged into      *
                               * the signal logging structure.      */
  }sigLogSignalPtrs;

  int_T         logFormat;          /* matrix=0, struct=1, or strut_wo_time=2 */

  int_T         logMaxRows;         /* Max number of rows (0 for no limit)    */
  int_T         logDecimation;      /* Data logging interval                  */

  const char_T  *logVarNameModifier;/* pre(post)fix string modifier for the   *
                                     * log variable names                     */

  const char_T  *logT;              /* Name of variable to log time           */
  const char_T  *logX;              /* Name of variable to log states         */
  const char_T  *logXFinal;         /* Name of varaible to log final state    */
  const char_T  *logY;              /* Name of variable(s) to log outputs     */
  const char_T  *logSL;          /* Name of variable(s) to log signal logging */

  union { /* Info about the states             */
      const RTWLogSignalInfo *cptr;
      RTWLogSignalInfo       *ptr;
  } logXSignalInfo;

  union {/* Info about the outptus            */
      const RTWLogSignalInfo *cptr;
      RTWLogSignalInfo       *ptr;
  }logYSignalInfo;

  union { /* Info about the sigLog signals   */
      const RTWLogSignalInfo *cptr;
      RTWLogSignalInfo       *ptr;
  } sigLogSignalInfo;

  void (*mdlLogData)(void *rtli, void *tPtr);

  const void * mmi;    /* Add the ModelMapping Info to the LogInfo
                        * so we can get at it for state logging */

} RTWLogInfo;

#endif

/* Macros associated with RTWLogInfo */
#define rtliGetLogInfo(rtli)     ((LogInfo*)(rtli)->logInfo)
#define rtliSetLogInfo(rtli,ptr) ((rtli)->logInfo = ((void *)ptr))

#define rtliGetLogFormat(rtli)   (rtli)->logFormat
#define rtliSetLogFormat(rtli,f) ((rtli)->logFormat = (f))

#define rtliGetLogVarNameModifier(rtli)      (rtli)->logVarNameModifier
#define rtliSetLogVarNameModifier(rtli,name) ((rtli)->logVarNameModifier=(name))

#define rtliGetLogMaxRows(rtli)     (rtli)->logMaxRows
#define rtliSetLogMaxRows(rtli,num) ((rtli)->logMaxRows = (num))

#define rtliGetLogDecimation(rtli)   (rtli)->logDecimation
#define rtliSetLogDecimation(rtli,l) ((rtli)->logDecimation = (l))

#define rtliGetLogT(rtli)     (rtli)->logT
#define rtliSetLogT(rtli,lt)  ((rtli)->logT = (lt))

#define rtliGetLogX(rtli)     (rtli)->logX
#define rtliSetLogX(rtli,lx)  ((rtli)->logX = (lx))

#define rtliGetLogY(rtli)     (rtli)->logY
#define rtliSetLogY(rtli,ly)  ((rtli)->logY = (ly))

#define rtliGetSigLog(rtli)     (rtli)->logSL
#define rtliSetSigLog(rtli,lsl)  ((rtli)->logSL = (lsl))

#define rtliGetLogXFinal(rtli)     (rtli)->logXFinal
#define rtliSetLogXFinal(rtli,lxf) ((rtli)->logXFinal = (lxf))

#define rtliGetLogXSignalInfo(rtli)     (rtli)->logXSignalInfo.cptr
#define rtliSetLogXSignalInfo(rtli,lxi) ((rtli)->logXSignalInfo.cptr = (lxi))
#define _rtliGetLogXSignalInfo(rtli)    (rtli)->logXSignalInfo.ptr

#define rtliGetLogYSignalInfo(rtli)     (rtli)->logYSignalInfo.cptr
#define rtliSetLogYSignalInfo(rtli,lyi) ((rtli)->logYSignalInfo.cptr = (lyi))
#define _rtliGetLogYSignalInfo(rtli)    (rtli)->logYSignalInfo.ptr

#define rtliGetSigLogSignalInfo(rtli)     (rtli)->sigLogSignalInfo.cptr
#define rtliSetSigLogSignalInfo(rtli,sli) ((rtli)->sigLogSignalInfo.cptr = (sli))
#define _rtliGetSigLogSignalInfo(rtli)    (rtli)->sigLogSignalInfo.ptr

#define rtliGetLogXSignalPtrs(rtli)     (rtli)->logXSignalPtrs.cptr
#define rtliSetLogXSignalPtrs(rtli,lxp) ((rtli)->logXSignalPtrs.cptr = (lxp))
#define _rtliGetLogXSignalPtrs(rtli)    (rtli)->logXSignalPtrs.ptr

#define rtliGetLogYSignalPtrs(rtli)     (rtli)->logYSignalPtrs.cptr
#define rtliSetLogYSignalPtrs(rtli,lyp) ((rtli)->logYSignalPtrs.cptr = (lyp))
#define _rtliGetLogYSignalPtrs(rtli)    (rtli)->logYSignalPtrs.ptr

#define rtliGetSigLogSignalPtrs(rtli)     (rtli)->sigLogSignalPtrs.cptr
#define rtliSetSigLogSignalPtrs(rtli,slp) ((rtli)->sigLogSignalPtrs.cptr = (slp))
#define _rtliGetSigLogSignalPtrs(rtli)    (rtli)->sigLogSignalPtrs.ptr

#define rtliGetMMI(rtli)     (rtli)->mmi
#define rtliSetMMI(rtli,mmiIn) ((rtli)->mmi = ((void *)mmiIn))

/* ========================================================================== */

#endif /* __RTW_MATLOGGING_H__ */
```

### rtw_modelmap.h
```c
/*
 * Copyright 1994-2010 The MathWorks, Inc.
 *
 * File: rtw_modelmap.h     $Revision: 1.1.6.3 $
 *
 * Abstract:
 *   Model tuning information.  Use the provided structure access methods
 *   whenever possible.
 *
 *   For details about these structures see Real-Time Workshop User's guide.
 */

#ifndef __RTW_MODELMAP__
#define __RTW_MODELMAP__

#ifdef SL_INTERNAL

# include "version.h"
# include "util.h"

#else

# include <stdlib.h>

#ifndef __RTW_UTFREE__
# define __RTW_UTFREE__
# define  utFree(arg)    if (arg) free(arg)
# define  utMalloc(arg)  malloc(arg)
#endif

#endif

#include <rtwtypes.h>
#include <rtw_capi.h>
#include <rtw_modelmap_logging.h>

typedef struct rtwCAPI_ModelMappingInfo_tag rtwCAPI_ModelMappingInfo;
typedef struct rtwCAPI_ModelMappingStaticInfo_tag rtwCAPI_ModelMappingStaticInfo;

/* ModelMappingStaticInfo */
struct rtwCAPI_ModelMappingStaticInfo_tag {
    /* signals */
    struct {
        rtwCAPI_Signals const *signals;     /* Signals Array */
        uint_T                numSignals;   /* Num Signals   */
        rtwCAPI_Signals const *rootInputs;  /* Root Inputs array */
        uint_T               numRootInputs; /* Num Root Inputs  */
        rtwCAPI_Signals const *rootOutputs; /* Root Outputs array */
        uint_T               numRootOutputs;/* Num Root Outputs  */
    } Signals;

    /* parameters */
    struct {
        rtwCAPI_BlockParameters const *blockParameters;   /* Block parameters Array   */
        uint_T                       numBlockParameters; /* Num block parameters     */
        rtwCAPI_ModelParameters const *modelParameters;   /* Model parameters Array*/
        uint_T                       numModelParameters; /* Num Model parameters  */
    } Params;

    /* states */
    struct {
        rtwCAPI_States const *states;   /* States array */
        uint_T               numStates; /* Num States   */
    } States;

    /* Static maps */
    /* datatypes, dimensions, fixed point, structure elements, sample times  */
    struct {
        rtwCAPI_DataTypeMap   const   *dataTypeMap;       /* Data Type Map          */
        rtwCAPI_DimensionMap  const   *dimensionMap;      /* Data Dimension Map     */
        rtwCAPI_FixPtMap      const   *fixPtMap;          /* Fixed Point Map        */
        rtwCAPI_ElementMap    const   *elementMap;        /* Structure Element map  */
        rtwCAPI_SampleTimeMap const   *sampleTimeMap;     /* Sample Times Map       */
        uint_T        const   *dimensionArray;    /* Dimension Array        */
    } Maps;

    /* TargetType - string specifying the intended target of the generated  *
     * C-API.                                                               *
     * targetType = "float"   - target supports floats and integer code     *
     *            = "integer" - target supports integer only code           */
    char_T const     *targetType;

    /* for internal use */
    rtwCAPI_ModelMapLoggingStaticInfo const *staticLogInfo;
};

/* ModelMappingInfo */
struct rtwCAPI_ModelMappingInfo_tag {
    /* ModelMappingInfo version */
    uint8_T                 versionNum;

    /* Reference to static model data, all model instances share this map   */
    rtwCAPI_ModelMappingStaticInfo *staticMap;

    /* Instance specific Maps, each model instance has a unique InstanceMap */
    struct {
        const char*                path;             /* Path to this instance */
        char*                      fullPath;
        void**                     dataAddrMap;      /* Data Address map      */
        rtwCAPI_ModelMappingInfo** childMMIArray;    /* array of child MMI    */
        uint_T                     childMMIArrayLen; /* Number of child MMIs  */
        int_T                      contStateStartIndex;  /* */

        /* for internal use */
        rtwCAPI_ModelMapLoggingInstanceInfo *instanceLogInfo;
        int32_T**                      vardimsAddrMap;   /* Vardims Address map   */
    } InstanceMap;
};

/* Macros for accessing ModelMappingStaticInfo fields */
#define rtwCAPI_GetSignalsFromStaticMap(SM)             ((SM)->Signals.signals)
#define rtwCAPI_GetNumSignalsFromStaticMap(SM)          ((SM)->Signals.numSignals)
#define rtwCAPI_GetLogSignalsArrayFromStaticMap(SM)     ((SM)->Signals.logSignalsArray)
#define rtwCAPI_GetNumLogSignalsFromStaticMap(SM)       ((SM)->Signals.numLogSignals)

#define rtwCAPI_GetBlockParametersFromStaticMap(SM)     ((SM)->Params.blockParameters)
#define rtwCAPI_GetNumBlockParametersFromStaticMap(SM)  ((SM)->Params.numBlockParameters)
#define rtwCAPI_GetModelParametersFromStaticMap(SM)     ((SM)->Params.modelParameters)
#define rtwCAPI_GetNumModelParametersFromStaticMap(SM)  ((SM)->Params.numModelParameters)

#define rtwCAPI_GetStatesFromStaticMap(SM)              ((SM)->States.states)
#define rtwCAPI_GetNumStatesFromStaticMap(SM)           ((SM)->States.numStates)

#define rtwCAPI_GetRootInputsFromStaticMap(SM)          ((SM)->Signals.rootInputs)
#define rtwCAPI_GetNumRootInputsFromStaticMap(SM)       ((SM)->Signals.numRootInputs)
#define rtwCAPI_GetRootOutputsFromStaticMap(SM)         ((SM)->Signals.rootOutputs)
#define rtwCAPI_GetNumRootOutputsFromStaticMap(SM)      ((SM)->Signals.numRootOutputs)

#define rtwCAPI_GetDataTypeMapFromStaticMap(SM)         ((SM)->Maps.dataTypeMap)
#define rtwCAPI_GetDimensionMapFromStaticMap(SM)        ((SM)->Maps.dimensionMap)
#define rtwCAPI_GetFixPtMapFromStaticMap(SM)            ((SM)->Maps.fixPtMap)
#define rtwCAPI_GetElementMapFromStaticMap(SM)          ((SM)->Maps.elementMap)
#define rtwCAPI_GetSampleTimeMapFromStaticMap(SM)       ((SM)->Maps.sampleTimeMap)
#define rtwCAPI_GetDimensionArrayFromStaticMap(SM)      ((SM)->Maps.dimensionArray)

/* Macros for accessing ModelMappingInfo fields */
#define rtwCAPI_GetSignals(MMI)         rtwCAPI_GetSignalsFromStaticMap((MMI)->staticMap)
#define rtwCAPI_GetNumSignals(MMI)      rtwCAPI_GetNumSignalsFromStaticMap((MMI)->staticMap)
#define rtwCAPI_GetLogSignalsArray(MMI) rtwCAPI_GetLogSignalsArrayFromStaticMap((MMI)->staticMap)
#define rtwCAPI_GetNumLogSignals(MMI)   rtwCAPI_GetNumLogSignalsFromStaticMap((MMI)->staticMap)

#define rtwCAPI_GetBlockParameters(MMI)    rtwCAPI_GetBlockParametersFromStaticMap((MMI)->staticMap)
#define rtwCAPI_GetNumBlockParameters(MMI) rtwCAPI_GetNumBlockParametersFromStaticMap((MMI)->staticMap)
#define rtwCAPI_GetModelParameters(MMI)    rtwCAPI_GetModelParametersFromStaticMap((MMI)->staticMap)
#define rtwCAPI_GetNumModelParameters(MMI) rtwCAPI_GetNumModelParametersFromStaticMap((MMI)->staticMap)

#define rtwCAPI_GetStates(MMI)     rtwCAPI_GetStatesFromStaticMap((MMI)->staticMap)
#define rtwCAPI_GetNumStates(MMI)  rtwCAPI_GetNumStatesFromStaticMap((MMI)->staticMap)

#define rtwCAPI_GetRootInputs(MMI)     rtwCAPI_GetRootInputsFromStaticMap((MMI)->staticMap)
#define rtwCAPI_GetNumRootInputs(MMI)  rtwCAPI_GetNumRootInputsFromStaticMap((MMI)->staticMap)
#define rtwCAPI_GetRootOutputs(MMI)    rtwCAPI_GetRootOutputsFromStaticMap((MMI)->staticMap)
#define rtwCAPI_GetNumRootOutputs(MMI) rtwCAPI_GetNumRootOutputsFromStaticMap((MMI)->staticMap)

#define rtwCAPI_GetDataTypeMap(MMI)       rtwCAPI_GetDataTypeMapFromStaticMap((MMI)->staticMap)
#define rtwCAPI_GetDimensionMap(MMI)      rtwCAPI_GetDimensionMapFromStaticMap((MMI)->staticMap)
#define rtwCAPI_GetFixPtMap(MMI)          rtwCAPI_GetFixPtMapFromStaticMap((MMI)->staticMap)
#define rtwCAPI_GetElementMap(MMI)        rtwCAPI_GetElementMapFromStaticMap((MMI)->staticMap)
#define rtwCAPI_GetSampleTimeMap(MMI)     rtwCAPI_GetSampleTimeMapFromStaticMap((MMI)->staticMap)
#define rtwCAPI_GetDimensionArray(MMI)    rtwCAPI_GetDimensionArrayFromStaticMap((MMI)->staticMap)

#define rtwCAPI_GetStaticLoggingInfo(MMI) ((MMI)->staticMap->staticLogInfo)

#define rtwCAPI_GetVersion(MMI)           ((MMI)->versionNum)
#define rtwCAPI_GetDataAddressMap(MMI)    ((MMI)->InstanceMap.dataAddrMap)
#define rtwCAPI_GetVarDimsAddressMap(MMI) ((MMI)->InstanceMap.vardimsAddrMap)
#define rtwCAPI_GetPath(MMI)              ((MMI)->InstanceMap.path)
#define rtwCAPI_GetFullPath(MMI)          ((MMI)->InstanceMap.fullPath)
#define rtwCAPI_GetChildMMI(MMI,i)        ((MMI)->InstanceMap.childMMIArray[i])
#define rtwCAPI_GetChildMMIArray(MMI)     ((MMI)->InstanceMap.childMMIArray)
#define rtwCAPI_GetChildMMIArrayLen(MMI)  ((MMI)->InstanceMap.childMMIArrayLen)
#define rtwCAPI_MMIGetContStateStartIndex(MMI) ((MMI)->InstanceMap.contStateStartIndex)
#define rtwCAPI_GetInstanceLoggingInfo(MMI) ((MMI)->InstanceMap.instanceLogInfo)

/* Macros for setting ModelMappingInfo fields */
#define rtwCAPI_SetVersion(MMI, n)            ((MMI).versionNum = (n))
#define rtwCAPI_SetStaticMap(MMI, statMap)    (MMI).staticMap = (statMap)
#define rtwCAPI_SetLoggingStaticMap(MMI,lStatMap) (MMI).staticMap->staticLogInfo = (lStatMap)
#define rtwCAPI_SetDataAddressMap(MMI, dAddr) (MMI).InstanceMap.dataAddrMap = (dAddr)
#define rtwCAPI_SetVarDimsAddressMap(MMI, vAddr) (MMI).InstanceMap.vardimsAddrMap = (vAddr)
#define rtwCAPI_SetPath(MMI,p)                (MMI).InstanceMap.path = (p)
#define rtwCAPI_SetFullPath(MMI,p)            (MMI).InstanceMap.fullPath = (p)
#define rtwCAPI_SetChildMMI(MMI,i,cMMI)       (MMI).InstanceMap.childMMIArray[i] = (cMMI)
#define rtwCAPI_SetChildMMIArray(MMI,cMMIs)   (MMI).InstanceMap.childMMIArray = (cMMIs)
#define rtwCAPI_SetChildMMIArrayLen(MMI,n)    (MMI).InstanceMap.childMMIArrayLen = (n)
#define rtwCAPI_MMISetContStateStartIndex(MMI,i) (MMI).InstanceMap.contStateStartIndex = (i)
#define rtwCAPI_SetInstanceLoggingInfo(MMI,l) (MMI).InstanceMap.instanceLogInfo = (l)

/* Functions in rtw_modelmap_utils.c */
#ifdef __cplusplus
extern "C" {
#endif
extern char* rtwCAPI_EncodePath(const char* path);
extern boolean_T rtwCAPI_HasStates(const rtwCAPI_ModelMappingInfo* mmi);
extern int_T rtwCAPI_GetNumStateRecords(const rtwCAPI_ModelMappingInfo* mmi);
extern int_T rtwCAPI_GetNumStateRecordsForRTWLogging(const rtwCAPI_ModelMappingInfo* mmi);
extern int_T rtwCAPI_GetNumContStateRecords(const rtwCAPI_ModelMappingInfo* mmi);
extern void  rtwCAPI_FreeFullPaths(rtwCAPI_ModelMappingInfo* mmi);
extern const char_T* rtwCAPI_UpdateFullPaths(rtwCAPI_ModelMappingInfo* mmi,
                                             const char_T*     path,
                                             boolean_T isCalledFromTopModel);
extern const char_T* rtwCAPI_GetStateRecordInfo(const rtwCAPI_ModelMappingInfo* mmi,
                                                const char_T**                  sigBlockName,
                                                const char_T**                  sigLabel,
                                                const char_T**                  sigName,
                                                int_T*                          sigWidth,
                                                int_T*                          sigDataType,
                                                int_T*                          logDataType,
                                                int_T*                          sigComplexity,
                                                void**                          sigDataAddr,
                                                boolean_T*                      sigCrossMdlRef,
                                                const char_T**                  sigPathAlias,
                                                double*                         sigSampleTime,
                                                int_T*                          sigIdx,
                                                boolean_T                       crossingModel,
                                                real_T*                         stateDerivVector,
                                                boolean_T                       rtwLogging);

extern int_T rtwCAPI_GetNumSigLogRecords(const rtwCAPI_ModelMappingInfo* mmi);
extern int_T rtwCAPI_GetNumSigLogRecordsForRTWLogging(const rtwCAPI_ModelMappingInfo* mmi);
extern const char_T* rtwCAPI_GetSigLogRecordInfo(const rtwCAPI_ModelMappingInfo* mmi,
                                                 const char_T**    sigBlockName,
                                                 const char_T**    sigLabel,
                                                 int_T*            sigWidth,
                                                 int_T*            sigDataType,
                                                 int_T*            logDataType,
                                                 int_T*            sigComplexity,
                                                 void**            sigDataAddr,
                                                 boolean_T*        sigCrossMdlRef,
                                                 int_T*            sigIdx,
                                                 boolean_T         crossingModel,
                                                 boolean_T         rtwLogging);

extern const char_T* rtwCAPI_GetFullContStateBlockPaths
(
    const rtwCAPI_ModelMappingInfo* mmi,
    char_T**                        blockPathsArray,
    size_t                          arrayLen,
    size_t                          startIndex,
    boolean_T                       crossingModel
    );

extern void rtwCAPI_CountSysRan(const rtwCAPI_ModelMappingInfo *mmi,
                                int                            *count);

extern void rtwCAPI_FillSysRan(const rtwCAPI_ModelMappingInfo *mmi,
			       sysRanDType                    **sysRan,
			       int                            *sysTid,
                               int                            *fillIdx);

#ifdef __cplusplus
}
#endif

#endif  /* __RTW_MODELMAP__ */

/* EOF - rtw_modelmap.h */
```

### rtw_modelmap_logging.h
```c
/*
 * Copyright 1994-2010 The MathWorks, Inc.
 *
 * File: rtw_modelmap_logging.h     $Revision: 1.1.6.3 $
 *
 * Abstract:
 *   Meta information used in conjunction with the ModelMappingInfo to
 *   facilitate logging.
 *
 */

#ifndef __RTW_MODELMAP_LOGGING__
#define __RTW_MODELMAP_LOGGING__

#include "sysran_types.h"

typedef struct rtwCAPI_ModelMapLoggingStaticInfo_tag rtwCAPI_ModelMapLoggingStaticInfo;
typedef struct rtwCAPI_ModelMapLoggingInstanceInfo_tag rtwCAPI_ModelMapLoggingInstanceInfo;

typedef struct rtwCAPI_LoggingMetaInfo_tag {
    uint_T sigIdx;   /* same index as the rtwCAPI_Signals */
    uint_T startIdx; /* starting index in the block I/O */
    const char *blockPath;
    uint_T portIdx;
    int_T  parentSysNum;   /* system number of the parent signal that requested
                              the logging */
} rtwCAPI_LoggingMetaInfo;

typedef enum {
    rtwCAPI_bus,
    rtwCAPI_signal
} rtwCAPI_LoggingBusElementType;

typedef struct rtwCAPI_LoggingBusElement_tag {
    uint_T                        index;
    rtwCAPI_LoggingBusElementType type;
} rtwCAPI_LoggingBusElement;

typedef struct rtwCAPI_LoggingBusSignals_tag {
    const char   *signalName;   /* logname should be in the sigProp */
    const char   *blockPath;
    uint_T  portIdx;
    uint_T  numElements;

    const rtwCAPI_LoggingBusElement *elements;
} rtwCAPI_LoggingBusSignals;

typedef struct rtwCAPI_StateflowSignalLoggingInfo_tag {
    const char   *signalName;
    const char   *blockPath;
    const char   *loggingName;
    uint_T       maxPoints;
    uint_T       decimation;
    boolean_T    useCustomName;
} rtwCAPI_StateflowSignalLoggingInfo;

/* Structure used for representing bus hierarchy information for dataset logging */
typedef struct rtwCAPI_SignalHierLoggingInfo_tag {
    const char_T* signalName;
    uint_T        numChildren;
    int_T         childStartIdx;
} rtwCAPI_SignalHierLoggingInfo;

typedef struct rtwCAPI_SignalHierLoggingInfoTable_tag {
    uint_T numSignals;
    rtwCAPI_SignalHierLoggingInfo const* infoTable;
    uint_T const* childIndexTable;
} rtwCAPI_SignalHierLoggingInfoTable;

/* ModelMapLoggingStaticInfo */
struct rtwCAPI_ModelMapLoggingStaticInfo_tag {
    /* Total number of non-virtual systems */
    uint_T numSystems;

    /* Effective context systems array */
    int_T const * contextSystems;

    rtwCAPI_LoggingMetaInfo const *logInfo;

    /* Bus signals info */
    uint_T numBusSignals;
    rtwCAPI_LoggingBusSignals const *busSignals;

    /* Dataset format hierarchy info */
    rtwCAPI_SignalHierLoggingInfoTable hierInfoTable;

    /* Dataset format Stateflow logging info */
    uint_T numChartSignals;
    rtwCAPI_StateflowSignalLoggingInfo const *chartSignals;
};

/* Macros for accessing static fields */
/* Note: These are all relative to the base MMI */
#define rtwCAPI_GetNumSystems(MMI) \
    ((MMI)->staticMap->staticLogInfo->numSystems)

#define rtwCAPI_GetContextSystems(MMI) \
    ((MMI)->staticMap->staticLogInfo->contextSystems)

#define rtwCAPI_GetLoggingInfoSigIdx(MMI, i) \
    ((MMI)->staticMap->staticLogInfo->logInfo[i].sigIdx)

#define rtwCAPI_GetLoggingInfoStartIdx(MMI, i) \
    ((MMI)->staticMap->staticLogInfo->logInfo[i].startIdx)

#define rtwCAPI_GetLoggingInfoBlockPath(MMI, i) \
    ((MMI)->staticMap->staticLogInfo->logInfo[i].blockPath)

#define rtwCAPI_GetLoggingInfoPortNumber(MMI, i) \
    ((MMI)->staticMap->staticLogInfo->logInfo[i].portIdx)

#define rtwCAPI_GetLoggingInfoParentSysNum(MMI, i) \
    ((MMI)->staticMap->staticLogInfo->logInfo[i].parentSysNum)

#define rtwCAPI_GetLoggingInfoNumBusSignals(MMI) \
    ((MMI)->staticMap->staticLogInfo->numBusSignals)

#define rtwCAPI_GetLoggingInfoBusSignalName(MMI, i) \
    ((MMI)->staticMap->staticLogInfo->busSignals[i].signalName)

#define rtwCAPI_GetLoggingInfoBusBlockPath(MMI, i) \
    ((MMI)->staticMap->staticLogInfo->busSignals[i].blockPath)

#define rtwCAPI_GetLoggingInfoBusPortIdx(MMI, i) \
    ((MMI)->staticMap->staticLogInfo->busSignals[i].portIdx)

#define rtwCAPI_GetLoggingInfoBusNumElements(MMI, i) \
    ((MMI)->staticMap->staticLogInfo->busSignals[i].numElements)

#define rtwCAPI_GetLoggingInfoBusElementIndex(MMI, i, j) \
    ((MMI)->staticMap->staticLogInfo->busSignals[i].elements[j].index)

#define rtwCAPI_GetLoggingInfoBusElementType(MMI, i, j) \
    ((MMI)->staticMap->staticLogInfo->busSignals[i].elements[j].type)

/* ModelMapLoggingInstanceInfo */
struct rtwCAPI_ModelMapLoggingInstanceInfo_tag {
    /* Pointer to the sysRan dwork pointers */
    sysRanDType **systemRan;

    /* Effective non-triggered tid of each system */
    int_T *systemTid;

    /* Points to the global tid map */
    int_T *globalTIDMap;
};

/* Note: These are all relative to the base MMI */

/* Get methods */
#define rtwCAPI_GetSystemRan(MMI) \
   ((MMI)->InstanceMap.instanceLogInfo->systemRan)

#define rtwCAPI_GetSystemTid(MMI) \
   ((MMI)->InstanceMap.instanceLogInfo->systemTid)

#define rtwCAPI_GetGlobalTIDMap(MMI) \
   ((MMI)->InstanceMap.instanceLogInfo->globalTIDMap)

/* Set methods */
#define rtwCAPI_SetSystemRan(MMI,s) \
   ((MMI).InstanceMap.instanceLogInfo->systemRan) = (s)

#define rtwCAPI_SetSystemTid(MMI,s) \
   ((MMI).InstanceMap.instanceLogInfo->systemTid) = (s)

#define rtwCAPI_SetGlobalTIDMap(MMI,s) \
   ((MMI).InstanceMap.instanceLogInfo->globalTIDMap) = (s)

#endif  /* __RTW_MODELMAP_LOGGING__ */

/* EOF - rtw_modelmap_logging.h */
```

### Library Logical/Libraries/J_IO_LIB (IEC, version 4.10.0)

#### J_IO_LIB.fun - Exported functions and function blocks
```iecst
(********************************************************************
 * COPYRIGHT -- INNIO Company
 ********************************************************************
 * Library: OutExist
 * File: OutExist.fun
 * Author: Schmid
 * Created: December 09, 2020
 ********************************************************************
 * Functions and function blocks of library OutExist
 ********************************************************************)

FUNCTION_BLOCK OutExist
	VAR_INPUT
		enable : BOOL;
		pPVstring : UDINT;
		pLastDatapoint : UDINT;
	END_VAR
	VAR_OUTPUT
		exist : BOOL;
		busy : BOOL;
		done : BOOL;
		pDatapoint : UDINT;
		sOutPVName : STRING[50];
	END_VAR
	VAR
		bSecondTry : BOOL;
		xAsIOFListDP : AsIOFListDP;
		xAsIOPVInfo : AsIOPVInfo;
		sPVstring : STRING[50];
		sPVfilter : STRING[60];
		bReadIOPVInfo : BOOL;
		pTempDatapoint : UDINT;
		zzEdge00000 : BOOL;
	END_VAR
END_FUNCTION_BLOCK
```

#### OutExist.st
```iecst
(********************************************************************

This code is confidential and proprietary to the INNIO Company.
It may not be used in any form, or reproduced in any manner, without the express
written permission of the INNIO Company.
Copyright, INNIO Company, 2021

Customized modifications: -
------------------------

History:
-------
V4.10	09-12-2020	Schmid,		initial version

Instructions for use:
--------------------
- Function can be used to check if an output variable is connected to the PLC

Outstandings: -
------------

*******************************************************************************)
FUNCTION_BLOCK OutExist

	IF EDGEPOS(enable) THEN			(* executed when enable triggered *)
		bSecondTry		:= FALSE;
		done			:= FALSE;
		bReadIOPVInfo	:= FALSE;
		pTempDatapoint	:= 0;
		brsstrcpy(ADR(sOutPVName), ADR(''));
	END_IF;

	IF NOT bSecondTry THEN
		(* create search string *)
		brsstrcpy(ADR(sPVfilter), ADR('/SourcePV='));
		IF pPVstring <> 0 THEN
			brsstrcpy(ADR(sPVstring), pPVstring);
		END_IF;
		brsstrcat(ADR(sPVfilter), ADR(sPVstring));
	END_IF;

	IF enable AND NOT done THEN
		(* get info on output variable from IOmap *)
		xAsIOFListDP.enable			:= NOT bReadIOPVInfo;
		xAsIOFListDP.pLastDatapoint	:= pLastDatapoint;
		xAsIOFListDP.flagsValue		:= 2#0000_0010_0010_0011;
		xAsIOFListDP.flagsMask		:= 2#0000_0011_0011_0011;
		xAsIOFListDP.pFilterString	:= ADR(sPVfilter);
		xAsIOFListDP();

		IF (xAsIOFListDP.status <> ERR_FUB_BUSY) AND xAsIOFListDP.enable THEN
			IF xAsIOFListDP.pDatapoint <> 0 THEN
				bReadIOPVInfo	:= TRUE;	(* datapoint found *)
				pTempDatapoint	:= xAsIOFListDP.pDatapoint;
			ELSE
				(* Second try with HalIO:: added to filter string *)
				brsstrcpy(ADR(sPVfilter), ADR('/SourcePV='));
				brsstrcpy(ADR(sPVstring), ADR('HalIO::'));
				IF pPVstring <> 0 THEN
					brsstrcat(ADR(sPVstring), pPVstring);
				END_IF;
				brsstrcat(ADR(sPVfilter), ADR(sPVstring));

				IF NOT bSecondTry AND NOT done THEN
					xAsIOFListDP();
				END_IF;

				bSecondTry := TRUE;

				IF xAsIOFListDP.status <> ERR_FUB_BUSY THEN
					IF xAsIOFListDP.pDatapoint <> 0 THEN
						bReadIOPVInfo	:= TRUE;	(* datapoint found *)
						pTempDatapoint	:= xAsIOFListDP.pDatapoint;
					ELSE
						(* no datapoint found *)
						exist			:= FALSE;
						pDatapoint		:= 0;
						brsstrcpy(ADR(sOutPVName), ADR(''));
						busy			:= FALSE;
						done			:= TRUE;
						bReadIOPVInfo	:= FALSE;
					END_IF;
				ELSE
					(* status busy *)
					busy			:= TRUE;
					done			:= FALSE;
					bReadIOPVInfo	:= FALSE;
				END_IF;
			END_IF;

		ELSIF (xAsIOFListDP.status = ERR_FUB_BUSY) THEN
			(* status busy *)
			busy			:= TRUE;
			done			:= FALSE;
			bReadIOPVInfo	:= FALSE;
		END_IF;

		(* Verify if found datapoint is correct *)
		xAsIOPVInfo.enable			:= bReadIOPVInfo;
		xAsIOPVInfo.index			:= 0;
		xAsIOPVInfo.pDatapoint		:= pTempDatapoint;
		xAsIOPVInfo();

		IF (xAsIOPVInfo.status <> ERR_FUB_BUSY) AND xAsIOPVInfo.enable THEN
			IF xAsIOPVInfo.pPvName <> 0 THEN
				IF strcmp(xAsIOPVInfo.pPvName, ADR(sPVstring)) = 0 THEN
					(* datapoint identical to search string *)
					exist		:= TRUE;
					pDatapoint	:= xAsIOFListDP.pDatapoint;
					brsstrcpy(ADR(sOutPVName), xAsIOPVInfo.pPvName);
				ELSE
					(* datapoint different to search string -> wrong datapoint found *)
					exist		:= FALSE;
					pDatapoint	:= 0;
					brsstrcpy(ADR(sOutPVName), ADR(''));
				END_IF;
			ELSE
				(* no name for datapoint found -> wrong datapoint found *)
				exist		:= FALSE;
				pDatapoint	:= 0;
				brsstrcpy(ADR(sOutPVName), ADR(''));
			END_IF;
			busy	:= FALSE;
			done	:= TRUE;
		ELSIF (xAsIOPVInfo.status = ERR_FUB_BUSY) THEN
			(* status busy *)
			busy	:= TRUE;
			done	:= FALSE;
		END_IF;

	ELSE
		(* disble FUBs after execution until retrigger via enable *)
		xAsIOFListDP.enable	:= FALSE;
		xAsIOPVInfo.enable	:= FALSE;
		bReadIOPVInfo		:= FALSE;
		pTempDatapoint		:= 0;
	END_IF;

END_FUNCTION_BLOCK
```

### Package Logical/AmmBase - AB: Alarm Management Base

### Data object Logical/AmmBase/META_AB (Simple) - MODUL META data file

#### META_AB.dat
```
; *******************************************************************************
; AGGR: Module Meta Data (data module)
;
; This code is confidential and proprietary to the INNIO Company.
; It may not be used in any form, or reproduced in any manner, without the express
; written permission of the INNIO Company.
; Copyright, INNIO Company, 2023
;
; Customized modifications: -
; ------------------------
;
; History:
; -------
; V03.99.00.00	06.03.2013	Weitzer		generated for modular software
;				29.05.2013	Zengerer	initial dependencies prepared
;				04.12.2013	lettenb.	dependencies added
; V04.00.00.00	31.01.2014	lettenb.	version + dependencies changed
; V04.00.02.00	17.06.2014	lettenb.	alarm test corr.
; V04.00.03.00	22.07.2014	lettenb.	para_task update, rem.reset logic corr.
; V04.03.00.00	02.03.2015	lettenb.	version + dependencies changed (920, CB added
; V04.03.01.00	02.11.2015	Zengerer 	MANDATORYMODULE statement
; V04.04.00.00	12.07.2016	Zengerer 	increase version number for changed customized array size
;               20.03.2017	lettenb.	remote reset from bus prepared, 3003(2103,2104) modif.acc.functional safety
;				07.08.2017	502413184	no shut down due TO a measuring signal failure, SWAT #3
; V04.05.00.00	22.12.2017	lettenb.	comment added: Safety-related application software source code (EN 13849-1 / 4.6.3)
; V04.05.01.00	08.03.2018	lettenb.	reset: 1056 bugfix
; V04.07.00.00	18.09.2018	lettenb.	iMsg declaration + library corrected
; V04.07.01.00	24.06.2019	Schmid		valid alarm number space for alarm test/bypass increased from 3999 to 9999
; V04.08.00.00	24.10.2019	Schmid		test bit for dry test bench added
; V04.11.00		02.02.2022	Denk		Group alarm for HMI internal warnings
; V04.12.00		25.01.2023	Perktold	AmmGnlTC5 created - derived from former parts of AmmGnl
; V04.13.00		04.12.2023	Bencze		Risk Class 10 for remote reset of safety trips
; V04.14.00		16.12.2024	Maran		bugfix: reset of temporary alarm bypass when the Service button is switched off (issue #1621)
;
; Instructions for use:
; --------------------
; make only changes at the version numbers
;
; Outstandings:
; ------------
;
; *******************************************************************************
;
"<META>"
;
; Module ID: 16961
"<MODUL>AB</MODUL>"
;
; Module Version (xx.yy.zz.cc)
"<VERSION>04.14.00.00</VERSION>"
;
; Module Basisupdate Version BU (00-99)
"<BASISUPDATE_VERSION>00</BASISUPDATE_VERSION>"
;
; Optional: specify order number for limitated module usage
"<ORDER></ORDER>" ;<!--(optional for restricted customizations; missing statement makes module valid for all orders)-->
;
; Parameter Check <PARAn Name='aAbcdef' MIN='xxx' MAX='yyy' />  (watch for correct spacings and apostrophs!)
"<PARAMETER_CHK>"
"<PARA1 Name='iEng_Motortype' MIN='208' MAX='920' />"
"<PARA2 Name='rN_EngStart_LimHi' MIN='50.0' MAX='2200.0' />"
"<PARA3 />"
"<PARA4 />"
"<PARA5 />"
"</PARAMETER_CHK>"
;
; Statement, if engine operation is also allowed without this module (FALSE) or if this module´s parameter check passing is mandatory (TRUE)
"<MANDATORYMODULE>TRUE</MANDATORYMODULE>"
;
; Permanent Datamodule Filenames<!-- NAME ist ohne Dateiendung einzutragen; Nur für Counter und interne Parameter verwenden-->
"<DATAMODULES>" ;<!-- optional; mehrere DATAMODULES erlaubt-->
"	<DATAMODULE>par_AB</DATAMODULE>"
"</DATAMODULES>"
;
; Dependencies Modules (MMxx.yy.zz.cc)
"<DEPENDENCIES>"
"	<DEPENDENCY MODULE='PB' VERSION='04.00.00.00' />"
"	<DEPENDENCY MODULE='HA' VERSION='04.00.00.00' />"
"	<DEPENDENCY MODULE='AG' VERSION='04.00.00.00' />"
"	<DEPENDENCY MODULE='CB' VERSION='04.03.00.00' />"
"	<DEPENDENCY MODULE='SY' VERSION='04.00.00.00' />"
"	<DEPENDENCY MODULE='OP' VERSION='04.00.00.00' />"
"	<DEPENDENCY MODULE='IG' VERSION='04.00.00.00' />"
"	<DEPENDENCY MODULE='HC' VERSION='04.00.00.00' />"
"	<DEPENDENCY MODULE='VE' VERSION='04.00.00.00' />"
"	<DEPENDENCY MODULE='VI' VERSION='04.11.00.00' />"
"	<DEPENDENCY MODULE='EX' VERSION='04.06.00.00' />"    ; corrected for SW download via HMI
"	<DEPENDENCY MODULE='TR' VERSION='04.05.00.00' />"    ; corrected for SW download via HMI
"	<DEPENDENCY MODULE='GC' VERSION='04.05.00.00' />"    ; corrected for SW download via HMI
"	<DEPENDENCY MODULE='CU' VERSION='04.06.00.00' />"    ; corrected for SW download via HMI
"	<DEPENDENCY MODULE='MO' VERSION='04.05.00.00' />"    ; corrected for SW download via HMI
"	<DEPENDENCY MODULE='IC' VERSION='04.05.00.00' />"    ; corrected for SW download via HMI
"	<DEPENDENCY MODULE='CP' VERSION='04.06.00.00' />"    ; corrected for SW download via HMI
"	<DEPENDENCY MODULE='EC' VERSION='04.06.00.00' />"    ; corrected for SW download via HMI
"	<DEPENDENCY MODULE='EG' VERSION='04.06.00.00' />"    ; corrected for SW download via HMI
"	<DEPENDENCY MODULE='KN' VERSION='04.06.00.00' />"    ; corrected for SW download via HMI
"	<DEPENDENCY MODULE='GM' VERSION='04.05.00.00' />"    ; corrected for SW download via HMI
"	<DEPENDENCY MODULE='GT' VERSION='04.06.00.00' />"    ; corrected for SW download via HMI
"	<DEPENDENCY MODULE='SA' VERSION='04.06.00.00' />"    ; corrected for SW download via HMI
"	<DEPENDENCY MODULE='KL' VERSION='04.06.00.00' />"    ; corrected for SW download via HMI
"	<DEPENDENCY MODULE='GD' VERSION='04.05.00.00' />"    ; corrected for SW download via HMI
"	<DEPENDENCY MODULE='CH' VERSION='04.06.00.00' />"    ; corrected for SW download via HMI
"	<DEPENDENCY MODULE='GR' VERSION='04.06.00.00' />"    ; corrected for SW download via HMI
"	<DEPENDENCY MODULE='EM' VERSION='04.06.00.00' />"    ; corrected for SW download via HMI
"	<DEPENDENCY VISVERSION='02.13.00.00' />" 			;Dependencies Visualization
"</DEPENDENCIES>"
;
; Module function description
"<MODULEFUNCTION>" ;<!-- short overview documentation of module function; add reference to detailed information, if available-->
"	<General>	"
"	Alarm management. "
"	</General>	"
""
"	<F1 Name='Alarm reset' LastModified='4.00.03.00'>"
"	Alarms reset, warnings reset, remote reset.	"
"	</F1>"
"	<F2 Name='Collect messages' LastModified='4.03.00.00'>"
"	Generation: general alarm, general warning, triptype 123.	"
"	</F2>"
"	<F3 Name='Alarm test' LastModified='4.03.00.00'>"
"	Alarm test mode control. Protection test function	"
"	</F3>"
""
"	<Info>"
"	UPDATE 4.07.00.00: iMsg size extended to 9999 "
"	</Info>"
""
"	<Customized LastModified='3.99.00.00'>"
"	- Nothing "
"	</Customized>	"
""
"</MODULEFUNCTION>"
;
"</META>"
```

### module_AB.typ
```iecst
TYPE
	IN_AB_Struct : 	STRUCT
		tPB2MM : ParaBase2MM_type;
		tVE2AB : MM2AmmBase; (*VE Ventilation*) (*OldName:newPv; Cycle:2;*)
		tHC2AB : MM2AmmBase; (*HC Heating Cooling*) (*OldName:newPv; Cycle:2;*)
		tEX2AB : MM2AmmBase; (*EX Exhaust*) (*OldName:newPv; Cycle:2;*)
		tTR2AB : MM2AmmBase; (*TR ThermalReactor*) (*OldName:newPv; Cycle:2;*)
		tGC2AB : MM2AmmBase; (*GC Generator Control*) (*OldName:newPv; Cycle:2;*)
		tCU2AB : MM2AmmBase; (*CU Customized*) (*OldName:newPv; Cycle:2;*)
		tMO2AB : MM2AmmBase; (*MO Monic*) (*OldName:newPv; Cycle:2;*)
		tIC2AB : MM2AmmBase; (*IC ICxxx*) (*OldName:newPv; Cycle:2;*)
		tIG2AB : MM2AmmBase; (*IG Ignition*) (*OldName:newPv; Cycle:2;*)
		tSY2AB : MM2AmmBase; (*SY Synchronization*) (*OldName:newPv; Cycle:2;*)
		tCP2AB : MM2AmmBase; (*CP Coupling*) (*OldName:newPv; Cycle:2;*)
		tEC2AB : MM2AmmBase; (*EC EngineController*) (*OldName:newPv; Cycle:2;*)
		tEG2AB : MM2AmmBase; (*EG EngineGeneral*) (*OldName:newPv; Cycle:2;*)
		tKN2AB : MM2AmmBase; (*KN Knocking*) (*OldName:newPv; Cycle:2;*)
		tGM2AB : MM2AmmBase; (*GM GasMixer*) (*OldName:newPv; Cycle:2;*)
		tGT2AB : MM2AmmBase; (*GT GasTrain*) (*OldName:newPv; Cycle:2;*)
		tAG2AB : MM2AmmBase; (*AG AuxiliariesGeneral*) (*OldName:newPv; Cycle:2;*)
		tOP2AB : MM2AmmBase; (*OP Opstate*) (*OldName:newPv; Cycle:2;*)
		tSA2AB : MM2AmmBase; (*SA SAFI*) (*OldName:newPv; Cycle:2;*)
		tKL2AB : MM2AmmBase; (*KL KLS98*) (*OldName:newPv; Cycle:2;*)
		tGD2AB : MM2AmmBase; (*GD GasMeteringUnit*) (*OldName:newPv; Cycle:2;*)
		tCH2AB : MM2AmmBase; (*CH ChargingUnit*) (*OldName:newPv; Cycle:2;*)
		tHA2AB : MM2AmmBase; (*HA HalIO*) (*OldName:newPv; Cycle:2;*)
		tPB2AB : MM2AmmBase; (*PB ParaBase*) (*OldName:newPv; Cycle:2;*)
		tTB2AB : MM2AmmBase; (*TB Test Bench*) (*OldName:newPv; Cycle:2;*)
		tVI2AB : MM2AmmBase; (*VI Visualization*) (*OldName:newPv; Cycle:2;*)
		tGR2AB : MM2AmmBase; (*GR GRidcode*) (*OldName:newPv; Cycle:2;*)
		tEM2AB : MM2AmmBase; (*EM emission*) (*OldName:newPv; Cycle:2;*)
		tCB2AB : MM2AmmBase; (*CB condition based management*) (*OldName:newPv; Cycle:2;*)
		tResetRemoteExt : HALioDi_Type; (*reset remote external*) (*OldName:E_FQUITT; Cycle:2;*)
		tGCB_On : HALioDi_Type; (*generator circuit breaker closed*) (*OldName:DI_GCB_ON; Cycle:2;*)
		tGCB_RUC : HALioDo_Type; (*generator circuit breaker release undervoltage coil*) (*OldName:DI_GCB_RUC; Cycle:2;*)
		tSafetyLoop_Eng : HALioDi_Type; (*safety loop engine*) (*OldName:SIS; Cycle:2;*)
		tEng_Run : HALioDo_Type; (*engine in operation*) (*OldName:BTRB; Cycle:2;*)
		iPassLevel : INT; (*pass level actual*) (*OldName:ucPassLevel; Cycle:2;*)
		iIdx_OMSS : INT; (*operation selection*) (*OldName:newPv; Cycle:2;*)
		iSt_OpMode : UDINT; (*engine operation status*) (*OldName:newPv; Cycle:2;*)
		rN_EngAct : REAL; (*engine speed actual [1/min]*) (*OldName:n_ist; Cycle:2;*)
		bEng_Start : BOOL; (*engine start*) (*OldName:M_STRT; Cycle:2*)
		bResetRemBus : BOOL; (* remote reset from fieldbus *) (*OldName:M_STRT; Cycle:5*)
		bMsg2101 : BOOL; (*signal failure engine cooling water temperature*) (*OldName:M_MSKWT; Cycle:2;*)
		bMsg2102 : BOOL; (*signal failure engine engine oil temperature*) (*OldName:M_MSOTP; Cycle:2;*)
		bMsg2103 : BOOL; (*signal failure engine engine oil pressure*) (*OldName:M_MSODR; Cycle:2;*)
		bMsg2104 : BOOL; (*signal failure engine engine cooling water pressure*) (*OldName:M_MSKWD; Cycle:2;*)
		bMsg3152 : BOOL; (*signal failure engine room air temperature*) (*OldName:M_MSRTM_W; Cycle:2;*)
		bGnlWarningHMI : BOOL; (*Internal HMI messsages for building group alarm*)
	END_STRUCT;
	OUT_AB_Struct : 	STRUCT
		tAB2PB : MM2ParaBase_type; (*AB Structure for this modules Para Services ( this is NOT tAB2PB! )*)
		tAB2VE : AmmBase2MM; (*VE Ventilation*) (*OldName:newPv; Cycle:2;*)
		tAB2HC : AmmBase2MM; (*HC Heating Cooling*) (*OldName:newPv; Cycle:2;*)
		tAB2EX : AmmBase2MM; (*EX Exhaust*) (*OldName:newPv; Cycle:2;*)
		tAB2TR : AmmBase2MM; (*TR ThermalReactor*) (*OldName:newPv; Cycle:2;*)
		tAB2GC : AmmBase2MM; (*GC Generator Control*) (*OldName:newPv; Cycle:2;*)
		tAB2CU : AmmBase2MM; (*CU Customized*) (*OldName:newPv; Cycle:2;*)
		tAB2MO : AmmBase2MM; (*MO Monic*) (*OldName:newPv; Cycle:2;*)
		tAB2IC : AmmBase2MM; (*IC ICxxx*) (*OldName:newPv; Cycle:2;*)
		tAB2IG : AmmBase2MM; (*IG Ignition*) (*OldName:newPv; Cycle:2;*)
		tAB2SY : AmmBase2MM; (*SY Synchronization*) (*OldName:newPv; Cycle:2;*)
		tAB2CP : AmmBase2MM; (*CP Coupling*) (*OldName:newPv; Cycle:2;*)
		tAB2EC : AmmBase2MM; (*EC EngineController*) (*OldName:newPv; Cycle:2;*)
		tAB2EG : AmmBase2MM; (*EG EngineGeneral*) (*OldName:newPv; Cycle:2;*)
		tAB2KN : AmmBase2MM; (*KN Knocking*) (*OldName:newPv; Cycle:2;*)
		tAB2GM : AmmBase2MM; (*GM GasMixer*) (*OldName:newPv; Cycle:2;*)
		tAB2GT : AmmBase2MM; (*GT GasTrain*) (*OldName:newPv; Cycle:2;*)
		tAB2AG : AmmBase2MM; (*AG AuxiliariesGeneral*) (*OldName:newPv; Cycle:2;*)
		tAB2OP : AmmBase2MM; (*OP Opstate*) (*OldName:newPv; Cycle:2;*)
		tAB2SA : AmmBase2MM; (*SA SAFI*) (*OldName:newPv; Cycle:2;*)
		tAB2KL : AmmBase2MM; (*KL KLS98*) (*OldName:newPv; Cycle:2;*)
		tAB2GD : AmmBase2MM; (*GD GasMeteringUnit*) (*OldName:newPv; Cycle:2;*)
		tAB2CH : AmmBase2MM; (*CH ChargingUnit*) (*OldName:newPv; Cycle:2;*)
		tAB2HA : AmmBase2MM; (*HA HalIO*) (*OldName:newPv; Cycle:2;*)
		tAB2GR : AmmBase2MM; (*GR GRidcode*) (*OldName:newPv; Cycle:2;*)
		tAB2EM : AmmBase2MM; (*EM emission*) (*OldName:newPv; Cycle:2;*)
		tAB2CB : AmmBase2MM; (*CB condition based management*) (*OldName:newPv; Cycle:2;*)
		tAlarmB2PB : AmmBase2MM; (*PB ParaBase( for AB data)*) (*OldName:newPv; Cycle:2;*)
		tAB2TB : AmmBase2MM; (*TB TestBench*) (*OldName:newPv; Cycle:2;*)
		tAB2VI : AmmBase2MM; (*VI Visualization*) (*OldName:newPv; Cycle:2;*)
		tResetWarning : HALioDo_Type; (*DO reset warning pulse*) (*OldName:DO_W_QUITT; Cycle:2;*)
		tResetTrip : HALioDo_Type; (*DO reset trip pulse*) (*OldName:DO_A_QUITT Cycle:2;*)
		tMonitoringOn : HALioDo_Type; (*DO monitoring on pulse(safety loop)*) (*OldName:UW_EIN; Cycle:2;*)
		tGnlTrip : HALioDo_Type; (*DO engine general trip*) (*OldName:A_SSTA; Cycle:2;*)
		tGnlWarning : HALioDo_Type; (*DO engine general warning*) (*OldName:A_SSTW; Cycle:2;*)
		bMsg3003 : BOOL; (*signal failure( 2101 or 2102 or 2103 or 2104 or 3152 > 24h)*) (*OldName:M_MS; Cycle:2;*)
		bServiceMode : BOOL; (*service mode*) (*OldName:bServiceBegin; Cycle:2;*)
		iMsg : ARRAY[0..9999]OF USINT; (*provides data from all alarms*) (*OldName:newPv; Cycle:2;*)
		bMMD_GenAlarmTestOn : BOOL; (*MMD_Gen alarm test On*) (*OldName:newPv; Cycle:2;*)
		bMMD_BB_AlarmTestOn : BOOL; (*MMD_BB  alarm test On*) (*OldName:newPv; Cycle:2;*)
	END_STRUCT;
	VIS2MM_Struct : 	STRUCT
		bResetLocVis : BOOL; (*reset local from vis*) (*OldName:E_QUITT; Cycle:5;*)
		bResetRemVis : BOOL; (*reset remote from vis*) (*OldName:VIS_FQUITT; Cycle:5;*)
		iNumAlarmTest : DINT; (*number alarm test from vis*) (*OldName:NumAmmTest; Cycle:5;*)
		bAlarmTestStart : BOOL; (*alarm test start from vis*) (*OldName:SetAmmTestStart; Cycle:5;*)
		bAlarmTestStop : BOOL; (*alarm test stop from vis*) (*OldName:SetAmmTestStop; Cycle:5;*)
		bServiceBegin : BOOL; (*service mode*) (*OldName:bServiceBegin; Cycle:5;*)
		bMMD_GenAlarmTestStart : BOOL; (*MMD_Gen alarm test start from vis*) (*OldName:newPv; Cycle:5;*)
		bMMD_GenAlarmTestStop : BOOL; (*MMD_Gen alarm test stop from vis*) (*OldName:newPv; Cycle:5;*)
		bMMD_BB_AlarmTestStart : BOOL; (*MMD_BB alarm test start from vis*) (*OldName:newPv; Cycle:5;*)
		bMMD_BB_AlarmTestStop : BOOL; (*MMD_BB alarm test stop from vis*) (*OldName:newPv; Cycle:5;*)
	END_STRUCT;
	MM2VIS_Struct : 	STRUCT
		bGnlTrip : BOOL; (*engine general trip*) (*OldName:M_SSTA; Cycle:5;*)
		bGnlTrip1 : BOOL; (*engine general trip 1*) (*OldName:M_SSTA1; Cycle:5;*)
		bGnlTrip2 : BOOL; (*engine general trip 2*) (*OldName:M_SSTA2; Cycle:5;*)
		bGnlTrip3 : BOOL; (*engine general trip 3*) (*OldName:M_SSTA3; Cycle:5;*)
		bGnlWarning : BOOL; (*engine general warning*) (*OldName:M_SSTW; Cycle:5;*)
		bTriptype1 : BOOL; (*triptype*) (*OldName:triptype_1; Cycle:5;*)
		bTriptype2 : BOOL; (*triptype*) (*OldName:triptype_2; Cycle:5;*)
		bTriptype3 : BOOL; (*triptype*) (*OldName:triptype_3; Cycle:5;*)
		bTriptypeS : BOOL; (*triptype*) (*OldName:RUHE; Cycle:5;*)
		bGnlTripDurEngOp : BOOL; (*engine general trip during engine operation*) (*OldName:newPv; Cycle:5;*)
		bAlarmTestEnable : BOOL; (*alarm test enable*) (*OldName:AmmTestEnable; Cycle:5;*)
		bNumAmmTestValid : BOOL; (*number alarm test valid*) (*OldName:NumAmmTestValid; Cycle:5;*)
		bAlarmTestOn : BOOL; (*alarm test On*) (*OldName:AmmTestOn; Cycle:5;*)
		iAlarmTestRestTime : INT; (*alarm test rest time [s]*) (*OldName:AmmTestRestTime; Cycle:5;*)
		bMMD_GenAlarmTestEnable : BOOL; (*MMD_Gen alarm test enable*) (*OldName:newPv; Cycle:5;*)
		bMMD_GenAlarmTestOn : BOOL; (*MMD_Gen alarm test On*) (*OldName:newPv; Cycle:5;*)
		iMMD_GenAlarmTestRestTime : INT; (*MMD_Gen alarm test rest time [s]*) (*OldName:newPv; Cycle:5;*)
		bMMD_BB_AlarmTestEnable : BOOL; (*MMD_BB alarm test enable*) (*OldName:newPv; Cycle:5;*)
		bMMD_BB_AlarmTestOn : BOOL; (*MMD_BB alarm test On*) (*OldName:newPv; Cycle:5;*)
		iMMD_BB_AlarmTestRestTime : INT; (*MMD_BB alarm test rest time [s]*) (*OldName:newPv; Cycle:5;*)
		bMsg1239 : BOOL; (*engine general trip*) (*OldName:M_SSTA; Cycle:5;*)
		bMsg1240 : BOOL; (*engine general warning*) (*OldName:M_SSTW; Cycle:5;*)
		bMsg1253 : BOOL; (*warm restart*) (*OldName:WARMSTART; Cycle:5;*)
		bMsg1254 : BOOL; (*cold restart*) (*OldName:KALTSTART; Cycle:5;*)
		bMsg1256 : BOOL; (*reset*) (*OldName:RM_QUITT; Cycle:5;*)
		bMsg3003 : BOOL; (*signal failure( 2101 or 2102 or 2103 or 2104 or 3152 > 24h)*) (*OldName:M_MS; Cycle:5;*)
		bMsg3252 : BOOL; (*remote reset*) (*OldName:T_FQUITT; Cycle:5;*)
		bMsg9389 : BOOL; (* W9389 Remote acknowledgement not possible, too many or safety trip *)
	END_STRUCT;
END_TYPE
```

### module_ABPara.typ
```iecst
TYPE
	PROGRAMMER_INFO : 	STRUCT
		DO_NOT_SORT_PARA : STRING[40] := 'DO NOT CHANGE PARAMETER SORTING!'; (*DO NOT CHANGE PARAMETER SORTING!*) (*ADD NEW PARAMETER ONLY AT THE END OF THE Para STRUCTURE. DO NOT DELETE existing Para items.*)
	END_STRUCT;
	Para_AB_struct : 	STRUCT
		iEng_Motortype : INT; (*Para motortype*) (*OldName:motortyp; Cycle:5;*)
		bVISA : BOOL; (*PARA [12259]: monitoring according VISA*) (*OldName:VISA; Cycle:5;*)
		rN_EngStart_LimHi : REAL; (*PARA [11296]: speed engine start limit high [1/min]*) (*OldName:GW_DREHZ; Cycle:5;*)
		rN_EngStart_HyHi : REAL; (*PARA [11295]: speed engine start limit high hysteresis [1/min]*) (*OldName:HY_DREHZ; Cycle:5;*)
		bResetRemActive : BOOL; (*PARA [10000]: remote reset active*) (*OldName:sel_rrActive; Cycle:5;*)
		iResetRemRiskClass : INT; (*PARA [10001]: remote reset risk class*) (*OldName:sel_rrClass; Cycle:5;*)
	END_STRUCT;
END_TYPE
```

### module_AB.var
```iecst
VAR
        bRemResWarning : BOOL := FALSE;
	bRemResIn : BOOL; (* remote reset is active *)
	xEngType : EngType; (*engine type*)
	xOpMode : OpMode; (*engine operation mode*)
	tMM2AB : MM2AmmBase; (*OUT: MM meta module AmmBase*) (*OldName:newPv; Cycle:2;*)
	tAB2MM : AmmBase2MM; (*IN:  AB AmmBase*) (*OldName:newPv; Cycle:2;*)
	IN_AB : IN_AB_Struct;
	OUT_AB : OUT_AB_Struct;
	MM2VIS : MM2VIS_Struct;
	VIS2MM : VIS2MM_Struct;
	Para : Para_AB_struct;
	ParaFactoryDefault : Para_AB_struct := (0); (*First Init Values*)
	pm : Para_AB_struct;
	bOMSS_Stop : BOOL; (*engine operation mode selection*)
	bOMSS_Man : BOOL; (*engine operation mode selection*)
	bOMSS_Aut : BOOL; (*engine operation mode selection*)
	bOMSS_Test : BOOL; (*engine operation mode selection*)
	bOMSS_Scav : BOOL; (*engine operation mode selection*)
	bOMSS_MAT : BOOL; (*engine operation mode selection*)
	bTriptype1 : BOOL; (*triptype*)
	bTriptype2 : BOOL; (*triptype*)
	bTriptype3 : BOOL; (*triptype*)
	bResetWarning : BOOL; (*reset warnings*)
	bResetTrip : BOOL; (*reset trip*)
	bGnlTrip : BOOL; (*general trip - common (project global)*)
	bGnlTrip1 : BOOL; (*general trip priority 1 - common (project global)*)
	bGnlTrip2 : BOOL; (*general trip priority 2 - common (project global)*)
	bGnlTrip3 : BOOL; (*general trip priority 3 - common (project global)*)
	bGnlWarning : BOOL; (*general warning - common (project global)*)
	bAlarmTestOn : BOOL; (*alarm test ON*)
	bAlarmTestEnable : BOOL; (*alarm test enable*)
	iAlarmTestRestTime : INT; (*alarm test rest time [s]*)
	iNumAlarmTestRun : DINT; (*number alarm test active*)
	bResetRiskClass0 : BOOL; (*reset risk class*)
	bResetRiskClass1 : BOOL; (*reset risk class*)
	bResetRiskClass2 : BOOL; (*reset risk class*)
	bResetRiskClass3 : BOOL; (*reset risk class*)
	bResetRiskClass4 : BOOL; (*reset risk class*)
	bRemResCmd : BOOL; (*remote reset command*)
	bN_EngStart : BOOL; (*engine start speed exceeded*)
	xTOF_ColdRestart : TOF := (0); (*cold restart*)
	xTOF_WarmRestart : TOF := (0); (*warm restart*)
	bNoInitDetected : BOOL := FALSE; (*allways true, except 1cycle on init up*)
	bWarmRestart : BOOL := (0); (*warm restart*)
	bColdRestart : BOOL := (0); (*cold restart*)
	bMMD_GenAlarmTestOn : BOOL; (*MMD_Gen alarm test ON*)
	bMMD_GenAlarmTestEnable : BOOL; (*MMD_Gen alarm test enable*)
	iMMD_GenAlarmTestRestTime : INT; (*MMD_Gen alarm test rest time [s]*)
	bMMD_BB_AlarmTestOn : BOOL; (*MMD_BB alarm test ON*)
	bMMD_BB_AlarmTestEnable : BOOL; (*MMD_BB alarm test enable*)
	iMMD_BB_AlarmTestRestTime : INT; (*MMD_BB alarm test rest time [s]*)
END_VAR
```

### Program Logical/AmmBase/default_AB (IEC, version 3.99.0) - values

#### default_ABCyclic.st
```iecst
(*******************************************************************************
default		value set

This code is confidential and proprietary to the INNIO Company.
It may not be used in any form, or reproduced in any manner,
without the express written permission of the INNIO Company.
Copyright, INNIO Company, 2019

Customized modifications: -
------------------------

History:
-------
V0.00.0	24.04.2012	lettenb.	new
V3.99.0	07.03.2013	lettenb.	cleanup

Instructions for use:
--------------------
Outstandings:
------------
*******************************************************************************)
PROGRAM _CYCLIC

	(* default TRUE setting for not existing Di's *)
//	IN_AB.x.Di		:=	IN_AB.x.Di		OR	NOT IN_AB.x.GoodQual;

END_PROGRAM
```

### Program Logical/AmmBase/general_AB (IEC, version 4.05.0) - functions

#### general_ABCyclic.st
```iecst
(*******************************************************************************
General		general functions

This code is confidential and proprietary to the INNIO Company.
It may not be used in any form, or reproduced in any manner,
without the express written permission of the INNIO Company.
Copyright, INNIO Company, 2019

Customized modifications: -
------------------------

History:
-------
V0.00.0	25.04.2012	lettenb.	new
V3.99.0	07.03.2013	lettenb.	cleanup
V4.05.0	31.10.2016				parameter check FOR diagnosis added

Instructions for use:
--------------------
Outstandings:
------------
*******************************************************************************)
PROGRAM _CYCLIC

	(* check para setup *)
	IN_AB.tPB2MM.bParaSetupOk;
	Para.iEng_Motortype;    (* MIN= 208   MAX= 920    *)
	Para.rN_EngStart_LimHi; (* MIN= 50.0  MAX= 2200.0 *)

	(* engine type defnition *)
	xEngType.Motortype := INT_TO_UINT(Para.iEng_Motortype);
	xEngType();

	(* engine operating mode selection *)
	bOMSS_Stop := FALSE;
	bOMSS_Man  := FALSE;
	bOMSS_Aut  := FALSE;
	bOMSS_Test := FALSE;
	bOMSS_Scav := FALSE;
	bOMSS_MAT  := FALSE;

	CASE IN_AB.iIdx_OMSS OF
	0:	bOMSS_Stop := TRUE;
	1:	bOMSS_Man  := TRUE;
		bOMSS_MAT  := TRUE;
	2:	bOMSS_Aut  := TRUE;
		bOMSS_MAT  := TRUE;
	3:	bOMSS_Test := TRUE;
		bOMSS_MAT  := TRUE;
	4:	bOMSS_Scav := TRUE;
	END_CASE;

	(* engine operating mode *)
	xOpMode(in:= IN_AB.iSt_OpMode);

	(* PLC Running *)
	IN_AB.tPB2MM.bSys_Run;

	(* engine start speed exceeded *)
	xGR_MAX_N_EngStart(In:= IN_AB.rN_EngAct, Gw:= Para.rN_EngStart_LimHi, Hy:= Para.rN_EngStart_HyHi);
	xTOF_N_EngStart(IN := xGR_MAX_N_EngStart.Q AND IN_AB.tPB2MM.bParaSetupOk, PT:= T#10s);
	bN_EngStart := xTOF_N_EngStart.Q;

END_PROGRAM
```

#### general_AB.var
```iecst
VAR
	xGR_MAX_N_EngStart : GR_MAXR;
	xTOF_N_EngStart : TOF;
END_VAR
```

### Program Logical/AmmBase/reset (IEC, version 4.13.0) - alarms
